C03630=1024.306,162.118,386.743,168.433,48.215,159.034
C03631=1024.301,161.869,386.765,168.430,48.220,159.035
C03632=1024.295,161.621,386.787,168.426,48.224,159.035
C03633=1024.290,161.372,386.809,168.423,48.229,159.036
C03634=1024.285,161.122,386.831,168.420,48.233,159.036
C03635=1024.279,160.874,386.853,168.417,48.238,159.037
C03636=1024.274,160.624,386.875,168.413,48.243,159.037
C03637=1024.269,160.375,386.897,168.410,48.247,159.037
C03638=1024.263,160.126,386.918,168.407,48.251,159.038
C03639=1024.258,159.878,386.941,168.403,48.256,159.038
C03640=1024.252,159.628,386.963,168.400,48.261,159.039
C03641=1024.247,159.380,386.985,168.397,48.265,159.039
C03642=1024.241,159.130,387.007,168.394,48.270,159.040
C03643=1024.236,158.882,387.028,168.391,48.275,159.040
C03644=1024.229,158.633,387.050,168.387,48.280,159.041
C03645=1024.225,158.383,387.071,168.384,48.285,159.041
C03646=1024.219,158.134,387.092,168.381,48.289,159.042
C03647=1024.213,157.886,387.114,168.378,48.294,159.042
C03648=1024.207,157.636,387.135,168.374,48.299,159.043
C03649=1024.202,157.388,387.157,168.371,48.303,159.043
C03650=1024.196,157.138,387.179,168.367,48.308,159.044
C03651=1024.190,156.890,387.200,168.365,48.313,159.044
C03652=1024.185,156.640,387.221,168.361,48.318,159.045
C03653=1024.179,156.392,387.242,168.358,48.322,159.045
C03654=1024.173,156.108,387.268,168.355,48.327,159.046
C03655=1024.166,155.825,387.292,168.350,48.333,159.046
C03656=1024.160,155.541,387.316,168.347,48.339,159.047
C03657=1024.153,155.258,387.340,168.343,48.344,159.047
C03658=1024.148,155.010,387.362,168.340,48.348,159.048
C03659=1024.142,154.760,387.383,168.337,48.353,159.048
C03660=1024.137,154.511,387.404,168.333,48.358,159.049
C03661=1024.131,154.262,387.426,168.330,48.363,159.049
C03662=1024.125,154.013,387.447,168.328,48.367,159.050
C03663=1024.119,153.764,387.468,168.324,48.372,159.050
C03664=1024.114,153.515,387.490,168.321,48.377,159.051
C03665=1024.109,153.266,387.511,168.317,48.382,159.051
C03666=1024.103,153.016,387.532,168.315,48.386,159.052
C03667=1024.098,152.768,387.554,168.311,48.391,159.052
C03668=1024.091,152.519,387.575,168.308,48.396,159.053
C03669=1024.086,152.270,387.596,168.305,48.401,159.053
C03670=1024.080,152.020,387.617,168.302,48.406,159.054
C03671=1024.074,151.772,387.639,168.299,48.411,159.054
C03672=1024.069,151.523,387.659,168.295,48.415,159.055
C03673=1024.063,151.274,387.681,168.292,48.420,159.055
C03674=1024.058,151.024,387.701,168.289,48.425,159.056
C03675=1024.052,150.775,387.723,168.286,48.430,159.056
C03676=1024.046,150.527,387.744,168.283,48.434,159.057
C03677=1024.041,150.278,387.765,168.279,48.439,159.057
C03678=1024.035,150.028,387.786,168.277,48.444,159.058
C03679=1024.029,149.779,387.807,168.273,48.449,159.058
C03680=1024.024,149.531,387.829,168.270,48.453,159.059
C03681=1024.019,149.281,387.850,168.266,48.458,159.059
C03682=1024.013,149.032,387.871,168.264,48.463,159.060
C03683=1024.008,148.783,387.892,168.260,48.468,159.060
C03684=1024.002,148.534,387.913,168.257,48.473,159.061
C03685=1023.996,148.285,387.934,168.255,48.477,159.061
C03686=1023.991,148.036,387.955,168.251,48.483,159.062
C03687=1023.985,147.786,387.976,168.248,48.487,159.063
C03688=1023.979,147.538,387.997,168.245,48.492,159.063
C03689=1023.974,147.289,388.018,168.242,48.497,159.064
C03690=1023.967,147.040,388.039,168.239,48.502,159.064
C03691=1023.962,146.791,388.059,168.235,48.506,159.065
C03692=1023.957,146.542,388.080,168.233,48.511,159.065
C03693=1023.951,146.292,388.102,168.229,48.516,159.066
C03694=1023.945,146.043,388.122,168.226,48.521,159.066
C03695=1023.940,145.795,388.143,168.224,48.525,159.067
C03696=1023.934,145.545,388.164,168.220,48.531,159.067
C03697=1023.929,145.296,388.185,168.217,48.536,159.068
C03698=1023.922,145.048,388.206,168.214,48.540,159.068
C03699=1023.917,144.799,388.226,168.211,48.545,159.069
C03700=1023.911,144.549,388.247,168.208,48.550,159.069
C03701=1023.906,144.300,388.268,168.204,48.555,159.070
C03702=1023.900,144.051,388.288,168.202,48.560,159.070
C03703=1023.894,143.802,388.309,168.199,48.565,159.071
C03704=1023.889,143.552,388.330,168.195,48.570,159.071
C03705=1023.883,143.303,388.350,168.192,48.574,159.072
C03706=1023.878,143.055,388.372,168.189,48.579,159.072
C03707=1023.871,142.805,388.392,168.186,48.584,159.073
C03708=1023.866,142.556,388.412,168.183,48.589,159.073
C03709=1023.861,142.307,388.433,168.181,48.594,159.074
C03710=1023.855,142.059,388.454,168.177,48.599,159.074
C03711=1023.848,141.809,388.475,168.174,48.604,159.075
C03712=1023.843,141.560,388.495,168.171,48.608,159.076
C03713=1023.838,141.311,388.516,168.168,48.613,159.076
C03714=1023.833,141.062,388.536,168.164,48.618,159.076
C03715=1023.826,140.813,388.557,168.162,48.623,159.077
C03716=1023.821,140.564,388.578,168.159,48.628,159.078
C03717=1023.815,140.315,388.598,168.155,48.633,159.078
C03718=1023.809,140.031,388.622,168.152,48.638,159.079
C03719=1023.802,139.748,388.645,168.149,48.644,159.079
C03720=1023.796,139.463,388.668,168.145,48.649,159.080
C03721=1023.790,139.180,388.692,168.142,48.655,159.080
C03722=1023.785,138.931,388.713,168.139,48.659,159.081
C03723=1023.779,138.682,388.733,168.136,48.664,159.081
C03724=1023.773,138.433,388.753,168.133,48.670,159.082
C03725=1023.768,138.184,388.774,168.130,48.674,159.083
C03726=1023.762,137.934,388.795,168.127,48.679,159.083
C03727=1023.756,137.686,388.815,168.123,48.684,159.084
C03728=1023.751,137.437,388.836,168.121,48.688,159.084
C03729=1023.745,137.188,388.856,168.118,48.694,159.085
C03730=1023.739,136.939,388.876,168.115,48.699,159.085
C03731=1023.733,136.690,388.896,168.112,48.703,159.086
C03732=1023.728,136.440,388.917,168.109,48.708,159.086
C03733=1023.723,136.190,388.937,168.106,48.714,159.087
C03734=1023.717,135.942,388.957,168.103,48.718,159.087
C03735=1023.711,135.693,388.978,168.100,48.723,159.088
C03736=1023.705,135.444,388.998,168.096,48.728,159.088
C03737=1023.700,135.195,389.018,168.094,48.733,159.089
C03738=1023.694,134.946,389.038,168.091,48.738,159.090
C03739=1023.688,134.696,389.059,168.087,48.743,159.090
C03740=1023.682,134.447,389.079,168.085,48.748,159.091
C03741=1023.677,134.198,389.099,168.082,48.753,159.091
C03742=1023.671,133.949,389.119,168.079,48.758,159.092
C03743=1023.666,133.700,389.140,168.076,48.763,159.092
C03744=1023.660,133.451,389.159,168.073,48.768,159.093
C03745=1023.655,133.202,389.180,168.070,48.772,159.093
C03746=1023.649,132.953,389.200,168.067,48.778,159.094
C03747=1023.644,132.704,389.220,168.064,48.783,159.094
C03748=1023.638,132.455,389.240,168.061,48.787,159.095
C03749=1023.632,132.205,389.261,168.058,48.792,159.095
C03750=1023.626,131.956,389.281,168.055,48.797,159.096
C03751=1023.621,131.706,389.301,168.053,48.802,159.097
C03752=1023.615,131.458,389.321,168.049,48.807,159.097
C03753=1023.609,131.208,389.341,168.047,48.812,159.098
C03754=1023.603,130.960,389.361,168.043,48.817,159.098
C03755=1023.598,130.711,389.382,168.040,48.822,159.099
C03756=1023.593,130.461,389.401,168.038,48.827,159.099
C03757=1023.587,130.212,389.421,168.034,48.832,159.100
C03758=1023.581,129.963,389.442,168.032,48.836,159.100
C03759=1023.576,129.714,389.461,168.029,48.842,159.101
C03760=1023.570,129.465,389.481,168.026,48.847,159.101
C03761=1023.564,129.216,389.501,168.023,48.851,159.102
C03762=1023.558,128.967,389.520,168.020,48.857,159.103
C03763=1023.553,128.718,389.541,168.017,48.862,159.103
C03764=1023.547,128.468,389.560,168.015,48.867,159.104
C03765=1023.540,128.219,389.580,168.011,48.872,159.104
C03766=1023.534,127.970,389.600,168.008,48.877,159.105
C03767=1023.529,127.720,389.619,168.006,48.882,159.105
C03768=1023.523,127.472,389.639,168.002,48.887,159.106
C03769=1023.517,127.222,389.659,167.999,48.892,159.106
C03770=1023.512,126.973,389.679,167.997,48.897,159.107
C03771=1023.506,126.724,389.698,167.994,48.902,159.108
C03772=1023.500,126.475,389.718,167.990,48.908,159.108
C03773=1023.494,126.225,389.738,167.988,48.912,159.109
C03774=1023.488,125.976,389.758,167.985,48.917,159.109
C03775=1023.483,125.727,389.777,167.982,48.923,159.110
C03776=1023.477,125.478,389.797,167.979,48.927,159.110
C03777=1023.471,125.229,389.817,167.976,48.932,159.111
C03778=1023.466,124.980,389.837,167.974,48.938,159.112
C03779=1023.460,124.730,389.856,167.970,48.942,159.112
C03780=1023.454,124.481,389.876,167.967,48.947,159.113
C03781=1023.448,124.232,389.895,167.965,48.953,159.113
C03782=1023.442,123.948,389.917,167.961,48.958,159.114
C03783=1023.435,123.665,389.940,167.958,48.964,159.114
C03784=1023.429,123.381,389.962,167.955,48.970,159.115
C03785=1023.422,123.097,389.984,167.952,48.975,159.116
C03786=1023.418,122.849,390.005,167.948,48.980,159.116
C03787=1023.412,122.600,390.024,167.946,48.985,159.117
C03788=1023.406,122.351,390.044,167.943,48.990,159.117
C03789=1023.400,122.101,390.063,167.939,48.995,159.118
C03790=1023.394,121.852,390.083,167.937,49.001,159.119
C03791=1023.389,121.603,390.102,167.934,49.005,159.119
C03792=1023.383,121.354,390.121,167.932,49.010,159.120
C03793=1023.377,121.105,390.141,167.928,49.015,159.120
C03794=1023.372,120.855,390.161,167.926,49.020,159.121
C03795=1023.366,120.606,390.180,167.923,49.025,159.121
C03796=1023.360,120.357,390.200,167.919,49.030,159.122
C03797=1023.355,120.107,390.220,167.917,49.035,159.122
C03798=1023.349,119.859,390.239,167.914,49.040,159.123
C03799=1023.343,119.610,390.259,167.912,49.045,159.123
C03800=1023.338,119.360,390.278,167.909,49.051,159.124
C03801=1023.332,119.112,390.298,167.906,49.055,159.125
C03802=1023.327,118.862,390.318,167.903,49.060,159.125
C03803=1023.321,118.612,390.337,167.900,49.065,159.126
C03804=1023.315,118.364,390.357,167.897,49.070,159.126
C03805=1023.309,118.114,390.376,167.894,49.075,159.127
C03806=1023.304,117.865,390.395,167.892,49.080,159.127
C03807=1023.299,117.616,390.414,167.888,49.085,159.128
C03808=1023.293,117.367,390.434,167.886,49.090,159.128
C03809=1023.287,117.118,390.453,167.883,49.095,159.129
C03810=1023.281,116.868,390.473,167.881,49.100,159.130
C03811=1023.276,116.619,390.493,167.877,49.104,159.130
C03812=1023.271,116.370,390.512,167.875,49.110,159.131
C03813=1023.265,116.121,390.531,167.872,49.115,159.131
C03814=1023.260,115.872,390.550,167.869,49.119,159.132
C03815=1023.254,115.623,390.570,167.866,49.124,159.132
C03816=1023.248,115.373,390.590,167.864,49.130,159.133
C03817=1023.243,115.125,390.609,167.861,49.135,159.133
C03818=1023.237,114.875,390.628,167.858,49.139,159.134
C03819=1023.231,114.626,390.647,167.855,49.144,159.134
C03820=1023.226,114.377,390.668,167.853,49.149,159.135
C03821=1023.220,114.127,390.687,167.849,49.154,159.136
C03822=1023.215,113.878,390.706,167.847,49.159,159.136
C03823=1023.210,113.629,390.725,167.844,49.164,159.137
C03824=1023.204,113.380,390.744,167.841,49.168,159.137
C03825=1023.198,113.131,390.764,167.838,49.174,159.138
C03826=1023.193,112.882,390.783,167.836,49.179,159.138
C03827=1023.187,112.633,390.802,167.833,49.184,159.139
C03828=1023.182,112.383,390.822,167.830,49.188,159.139
C03829=1023.176,112.134,390.841,167.827,49.194,159.140
C03830=1023.170,111.884,390.860,167.825,49.199,159.140
C03831=1023.165,111.636,390.879,167.821,49.203,159.141
C03832=1023.159,111.386,390.898,167.819,49.209,159.142
C03833=1023.153,111.137,390.917,167.816,49.214,159.142
C03834=1023.147,110.888,390.936,167.814,49.219,159.143
C03835=1023.142,110.639,390.955,167.811,49.224,159.143
C03836=1023.137,110.389,390.974,167.808,49.229,159.144
C03837=1023.131,110.140,390.993,167.805,49.234,159.144
C03838=1023.124,109.891,391.012,167.802,49.239,159.145
C03839=1023.119,109.642,391.031,167.800,49.244,159.145
C03840=1023.114,109.393,391.050,167.797,49.249,159.146
C03841=1023.107,109.144,391.069,167.794,49.254,159.147
C03842=1023.102,108.894,391.088,167.791,49.260,159.147
C03843=1023.097,108.645,391.106,167.789,49.264,159.148
C03844=1023.090,108.396,391.125,167.785,49.269,159.148
C03845=1023.085,108.146,391.144,167.783,49.275,159.149
C03846=1023.078,107.862,391.166,167.779,49.281,159.150
C03847=1023.072,107.579,391.187,167.776,49.286,159.150
C03848=1023.065,107.295,391.209,167.773,49.292,159.151
C03849=1023.058,107.011,391.230,167.770,49.298,159.151
C03850=1023.053,106.762,391.249,167.767,49.303,159.152
C03851=1023.047,106.513,391.267,167.765,49.308,159.153
C03852=1023.041,106.264,391.286,167.762,49.313,159.153
C03853=1023.036,106.014,391.306,167.760,49.318,159.154
C03854=1023.030,105.765,391.323,167.756,49.323,159.154
C03855=1023.024,105.516,391.343,167.754,49.328,159.155
C03856=1023.018,105.267,391.361,167.751,49.333,159.155
C03857=1023.013,105.018,391.380,167.749,49.339,159.156
C03858=1023.008,104.768,391.399,167.746,49.344,159.157
C03859=1023.001,104.519,391.417,167.743,49.348,159.157
C03860=1022.996,104.270,391.436,167.740,49.354,159.158
C03861=1022.990,104.021,391.455,167.738,49.359,159.158
C03862=1022.984,103.771,391.473,167.734,49.364,159.159
C03863=1022.979,103.522,391.492,167.731,49.369,159.159
C03864=1022.973,103.273,391.511,167.729,49.374,159.160
C03865=1022.967,103.024,391.530,167.726,49.379,159.160
C03866=1022.962,102.774,391.548,167.724,49.384,159.161
C03867=1022.956,102.525,391.567,167.721,49.389,159.162
C03868=1022.950,102.276,391.586,167.718,49.394,159.162
C03869=1022.945,102.027,391.605,167.716,49.399,159.163
C03870=1022.939,101.777,391.623,167.713,49.404,159.163
C03871=1022.934,101.529,391.642,167.710,49.409,159.164
C03872=1022.927,101.279,391.660,167.707,49.414,159.165
C03873=1022.922,101.029,391.679,167.705,49.419,159.165
C03874=1022.917,100.781,391.698,167.702,49.424,159.166
C03875=1022.910,100.532,391.717,167.700,49.429,159.166
C03876=1022.906,100.282,391.735,167.696,49.434,159.167
C03877=1022.900,100.033,391.754,167.694,49.439,159.167
C03878=1022.894,99.783,391.772,167.691,49.445,159.168
C03879=1022.889,99.534,391.791,167.689,49.449,159.168
C03880=1022.882,99.285,391.809,167.685,49.454,159.169
C03881=1022.877,99.035,391.828,167.683,49.460,159.170
C03882=1022.871,98.787,391.846,167.680,49.465,159.170
C03883=1022.865,98.537,391.864,167.678,49.470,159.171
C03884=1022.860,98.288,391.883,167.675,49.475,159.171
C03885=1022.854,98.039,391.901,167.673,49.480,159.172
C03886=1022.847,97.789,391.920,167.669,49.485,159.172
C03887=1022.843,97.540,391.938,167.666,49.490,159.173
C03888=1022.836,97.291,391.956,167.664,49.496,159.174
C03889=1022.831,97.042,391.974,167.661,49.501,159.174
C03890=1022.825,96.792,391.992,167.659,49.506,159.175
C03891=1022.819,96.543,392.011,167.655,49.511,159.175
C03892=1022.813,96.294,392.029,167.653,49.516,159.176
C03893=1022.808,96.044,392.048,167.650,49.521,159.176
C03894=1022.802,95.795,392.066,167.648,49.526,159.177
C03895=1022.796,95.546,392.084,167.645,49.532,159.178
C03896=1022.791,95.297,392.102,167.642,49.536,159.178
C03897=1022.785,95.047,392.120,167.639,49.542,159.179
C03898=1022.779,94.799,392.139,167.637,49.547,159.179
C03899=1022.774,94.548,392.157,167.634,49.552,159.180
C03900=1022.768,94.300,392.175,167.632,49.557,159.181
C03901=1022.762,94.050,392.193,167.628,49.562,159.181
C03902=1022.756,93.801,392.211,167.626,49.567,159.182
C03903=1022.750,93.552,392.230,167.623,49.572,159.182
C03904=1022.745,93.303,392.248,167.621,49.577,159.183
C03905=1022.739,93.053,392.266,167.618,49.583,159.183
C03906=1022.734,92.804,392.284,167.616,49.587,159.184
C03907=1022.728,92.555,392.302,167.612,49.592,159.184
C03908=1022.722,92.306,392.321,167.610,49.598,159.185
C03909=1022.716,92.056,392.339,167.607,49.603,159.185
C03910=1022.710,91.773,392.360,167.604,49.608,159.186
C03911=1022.703,91.488,392.380,167.601,49.614,159.187
C03912=1022.697,91.205,392.401,167.598,49.620,159.187
C03913=1022.691,90.922,392.421,167.595,49.625,159.188
C03914=1022.684,90.672,392.439,167.593,49.631,159.189
C03915=1022.679,90.423,392.458,167.590,49.636,159.189
C03916=1022.673,90.174,392.476,167.587,49.640,159.190
C03917=1022.668,89.925,392.494,167.584,49.646,159.190
C03918=1022.662,89.674,392.512,167.582,49.651,159.191
C03919=1022.657,89.426,392.531,167.579,49.656,159.191
C03920=1022.651,89.177,392.548,167.577,49.661,159.192
C03921=1022.645,88.927,392.566,167.573,49.666,159.193
C03922=1022.639,88.678,392.584,167.571,49.672,159.193
C03923=1022.633,88.428,392.602,167.568,49.677,159.194
C03924=1022.628,88.179,392.619,167.566,49.682,159.194
C03925=1022.622,87.930,392.637,167.563,49.687,159.195
C03926=1022.616,87.681,392.655,167.561,49.692,159.196
C03927=1022.610,87.432,392.673,167.558,49.697,159.196
C03928=1022.604,87.183,392.691,167.555,49.702,159.197
C03929=1022.598,86.933,392.709,167.552,49.708,159.197
C03930=1022.593,86.684,392.726,167.550,49.712,159.198
C03931=1022.587,86.435,392.744,167.547,49.718,159.198
C03932=1022.581,86.185,392.762,167.545,49.723,159.199
C03933=1022.575,85.936,392.779,167.542,49.728,159.200
C03934=1022.569,85.686,392.797,167.539,49.733,159.200
C03935=1022.564,85.437,392.815,167.536,49.739,159.201
C03936=1022.558,85.187,392.833,167.534,49.744,159.201
C03937=1022.552,84.938,392.850,167.531,49.749,159.202
C03938=1022.547,84.689,392.868,167.529,49.754,159.202
C03939=1022.540,84.440,392.886,167.526,49.759,159.203
C03940=1022.535,84.191,392.903,167.524,49.764,159.204
C03941=1022.529,83.941,392.921,167.520,49.769,159.204
C03942=1022.523,83.692,392.939,167.518,49.774,159.205
C03943=1022.518,83.443,392.957,167.515,49.780,159.205
C03944=1022.512,83.193,392.974,167.513,49.784,159.206
C03945=1022.506,82.944,392.992,167.510,49.790,159.206
C03946=1022.501,82.695,393.010,167.508,49.795,159.207
C03947=1022.495,82.445,393.028,167.504,49.800,159.207
C03948=1022.489,82.196,393.045,167.502,49.805,159.208
C03949=1022.483,81.947,393.063,167.499,49.810,159.209
C03950=1022.477,81.697,393.081,167.497,49.816,159.209
C03951=1022.472,81.448,393.098,167.494,49.821,159.210
C03952=1022.466,81.199,393.116,167.491,49.825,159.210
C03953=1022.460,80.950,393.134,167.489,49.831,159.211
C03954=1022.455,80.700,393.151,167.486,49.836,159.211
C03955=1022.449,80.451,393.169,167.484,49.841,159.212
C03956=1022.443,80.202,393.187,167.481,49.846,159.213
C03957=1022.438,79.952,393.204,167.479,49.851,159.213
C03958=1022.432,79.703,393.221,167.475,49.856,159.214
C03959=1022.426,79.453,393.239,167.473,49.861,159.214
C03960=1022.421,79.204,393.257,167.470,49.866,159.215
C03961=1022.415,78.955,393.274,167.468,49.871,159.215
C03962=1022.409,78.705,393.292,167.465,49.877,159.216
C03963=1022.404,78.456,393.310,167.463,49.882,159.216
C03964=1022.398,78.207,393.327,167.460,49.886,159.217
C03965=1022.392,77.958,393.345,167.457,49.891,159.217
C03966=1022.387,77.708,393.362,167.455,49.897,159.218
C03967=1022.381,77.459,393.380,167.452,49.902,159.219
C03968=1022.376,77.210,393.397,167.449,49.906,159.219
C03969=1022.369,76.960,393.415,167.446,49.912,159.220
C03970=1022.364,76.711,393.431,167.444,49.917,159.220
C03971=1022.358,76.462,393.449,167.441,49.923,159.221
C03972=1022.353,76.213,393.467,167.439,49.927,159.222
C03973=1022.346,75.963,393.484,167.436,49.932,159.222
C03974=1022.340,75.679,393.504,167.433,49.939,159.223
C03975=1022.333,75.396,393.524,167.430,49.945,159.223
C03976=1022.327,75.112,393.543,167.427,49.950,159.224
C03977=1022.320,74.828,393.562,167.424,49.956,159.225
C03978=1022.314,74.579,393.580,167.421,49.962,159.225
C03979=1022.309,74.330,393.597,167.419,49.966,159.226
C03980=1022.302,74.080,393.614,167.417,49.971,159.226
C03981=1022.297,73.831,393.632,167.414,49.977,159.227
C03982=1022.292,73.582,393.649,167.411,49.982,159.228
C03983=1022.285,73.333,393.666,167.409,49.987,159.228
C03984=1022.279,73.083,393.684,167.406,49.992,159.229
C03985=1022.274,72.833,393.700,167.403,49.997,159.229
C03986=1022.268,72.584,393.718,167.401,50.003,159.230
C03987=1022.262,72.335,393.734,167.398,50.008,159.230
C03988=1022.256,72.085,393.752,167.395,50.012,159.231
C03989=1022.251,71.836,393.770,167.393,50.018,159.231
C03990=1022.245,71.587,393.786,167.390,50.023,159.232
C03991=1022.239,71.338,393.803,167.387,50.028,159.232
C03992=1022.234,71.088,393.820,167.385,50.033,159.233
C03993=1022.227,70.839,393.838,167.382,50.038,159.234
C03994=1022.222,70.589,393.855,167.380,50.044,159.234
C03995=1022.217,70.340,393.872,167.377,50.049,159.235
C03996=1022.211,70.091,393.888,167.374,50.053,159.235
C03997=1022.205,69.842,393.906,167.372,50.059,159.236
C03998=1022.200,69.593,393.923,167.369,50.064,159.236
C03999=1022.193,69.343,393.940,167.367,50.069,159.237
C04000=1022.188,69.094,393.958,167.364,50.074,159.238
C04001=1022.182,68.844,393.975,167.362,50.079,159.238
C04002=1022.176,68.595,393.992,167.358,50.084,159.239
C04003=1022.171,68.346,394.008,167.356,50.090,159.239
C04004=1022.164,68.095,394.025,167.353,50.095,159.240
C04005=1022.159,67.846,394.043,167.351,50.099,159.240
C04006=1022.153,67.597,394.059,167.348,50.105,159.241
C04007=1022.147,67.348,394.076,167.346,50.110,159.242
C04008=1022.141,67.099,394.093,167.343,50.116,159.242
C04009=1022.136,66.850,394.110,167.340,50.120,159.243
C04010=1022.130,66.600,394.126,167.337,50.125,159.243
C04011=1022.124,66.350,394.144,167.335,50.131,159.244
C04012=1022.118,66.101,394.161,167.332,50.136,159.244
C04013=1022.113,65.852,394.177,167.330,50.141,159.245
C04014=1022.107,65.602,394.194,167.327,50.146,159.245
C04015=1022.101,65.353,394.211,167.325,50.151,159.246
C04016=1022.095,65.104,394.228,167.323,50.157,159.247
C04017=1022.090,64.854,394.244,167.319,50.162,159.247
C04018=1022.084,64.605,394.261,167.317,50.166,159.248
C04019=1022.078,64.355,394.279,167.314,50.172,159.248
C04020=1022.072,64.106,394.295,167.312,50.177,159.249
C04021=1022.066,63.857,394.312,167.309,50.182,159.249
C04022=1022.060,63.607,394.329,167.307,50.187,159.250
C04023=1022.055,63.358,394.346,167.303,50.193,159.250
C04024=1022.049,63.108,394.362,167.301,50.197,159.251
C04025=1022.043,62.860,394.379,167.298,50.203,159.252
C04026=1022.037,62.610,394.395,167.296,50.208,159.252
C04027=1022.031,62.360,394.412,167.293,50.214,159.253
C04028=1022.025,62.111,394.429,167.291,50.218,159.253
C04029=1022.019,61.861,394.445,167.288,50.224,159.254
C04030=1022.013,61.612,394.461,167.285,50.229,159.254
C04031=1022.007,61.362,394.477,167.283,50.235,159.255
C04032=1022.001,61.114,394.494,167.280,50.240,159.256
C04033=1021.996,60.864,394.511,167.278,50.245,159.256
C04034=1021.990,60.615,394.527,167.274,50.250,159.257
C04035=1021.984,60.365,394.544,167.273,50.256,159.257
C04036=1021.978,60.116,394.560,167.269,50.261,159.258
C04037=1021.972,59.867,394.576,167.267,50.266,159.259
C04038=1021.965,59.549,394.597,167.264,50.273,159.259
C04039=1021.957,59.232,394.618,167.260,50.280,159.260
C04040=1021.950,58.915,394.638,167.257,50.287,159.261
C04041=1021.942,58.598,394.660,167.254,50.293,159.262
C04042=1021.937,58.348,394.677,167.251,50.298,159.262
C04043=1021.931,58.099,394.693,167.248,50.304,159.263
C04044=1021.924,57.849,394.710,167.246,50.309,159.263
C04045=1021.918,57.599,394.726,167.242,50.314,159.264
C04046=1021.912,57.350,394.742,167.241,50.319,159.264
C04047=1021.906,57.101,394.758,167.237,50.324,159.265
C04048=1021.900,56.851,394.775,167.235,50.330,159.265
C04049=1021.895,56.602,394.791,167.232,50.335,159.266
C04050=1021.889,56.352,394.808,167.230,50.340,159.266
C04051=1021.883,56.103,394.824,167.227,50.345,159.267
C04052=1021.877,55.854,394.840,167.225,50.350,159.268
C04053=1021.871,55.604,394.856,167.222,50.356,159.268
C04054=1021.865,55.355,394.873,167.220,50.361,159.269
C04055=1021.859,55.106,394.889,167.216,50.366,159.269
C04056=1021.854,54.856,394.906,167.215,50.371,159.270
C04057=1021.848,54.607,394.922,167.211,50.376,159.270
C04058=1021.843,54.358,394.938,167.209,50.381,159.271
C04059=1021.837,54.109,394.954,167.206,50.387,159.271
C04060=1021.831,53.859,394.970,167.204,50.392,159.272
C04061=1021.825,53.609,394.986,167.201,50.397,159.273
C04062=1021.819,53.360,395.002,167.199,50.402,159.273
C04063=1021.813,53.111,395.019,167.196,50.407,159.274
C04064=1021.808,52.861,395.035,167.194,50.413,159.274
C04065=1021.802,52.612,395.052,167.190,50.418,159.275
C04066=1021.796,52.362,395.068,167.188,50.423,159.275
C04067=1021.790,52.113,395.084,167.185,50.428,159.276
C04068=1021.784,51.864,395.100,167.183,50.433,159.276
C04069=1021.778,51.614,395.117,167.180,50.438,159.277
C04070=1021.774,51.381,395.132,167.178,50.443,159.277
C04071=1021.768,51.149,395.147,167.175,50.448,159.278
C04072=1021.763,50.916,395.162,167.173,50.453,159.278
C04073=1021.757,50.684,395.177,167.171,50.457,159.279
C04074=1021.752,50.450,395.192,167.169,50.462,159.280
C04075=1021.747,50.218,395.207,167.165,50.467,159.280
C04076=1021.742,49.985,395.222,167.163,50.472,159.280
C04077=1021.736,49.752,395.237,167.161,50.476,159.281
C04078=1021.730,49.503,395.253,167.159,50.482,159.282
C04079=1021.725,49.254,395.269,167.155,50.487,159.282
C04080=1021.719,49.005,395.286,167.153,50.492,159.283
C04081=1021.713,48.756,395.302,167.150,50.497,159.283
C04082=1021.708,48.505,395.318,167.148,50.502,159.284
C04083=1021.702,48.256,395.334,167.145,50.507,159.284
C04084=1021.696,48.007,395.350,167.143,50.512,159.285
C04085=1021.690,47.757,395.367,167.140,50.517,159.285
C04086=1021.684,47.509,395.383,167.137,50.523,159.286
C04087=1021.679,47.259,395.398,167.135,50.527,159.286
C04088=1021.673,47.009,395.414,167.132,50.533,159.287
C04089=1021.667,46.760,395.431,167.130,50.537,159.287
C04090=1021.661,46.511,395.447,167.127,50.542,159.288
C04091=1021.656,46.260,395.463,167.125,50.548,159.288
C04092=1021.651,46.012,395.479,167.122,50.553,159.289
C04093=1021.645,45.762,395.495,167.119,50.558,159.289
C04094=1021.639,45.513,395.511,167.117,50.563,159.290
C04095=1021.633,45.263,395.527,167.114,50.568,159.290
C04096=1021.627,45.014,395.543,167.112,50.572,159.291
C04097=1021.622,44.765,395.559,167.109,50.578,159.292
C04098=1021.616,44.516,395.575,167.106,50.583,159.292
C04099=1021.610,44.266,395.591,167.104,50.588,159.293
C04100=1021.604,44.016,395.607,167.101,50.593,159.293
C04101=1021.599,43.767,395.624,167.099,50.598,159.294
C04102=1021.593,43.483,395.641,167.096,50.604,159.294
C04103=1021.586,43.199,395.660,167.093,50.609,159.295
C04104=1021.580,42.914,395.678,167.090,50.615,159.295
C04105=1021.574,42.631,395.696,167.087,50.620,159.296
C04106=1021.568,42.382,395.713,167.084,50.626,159.296
C04107=1021.562,42.132,395.728,167.082,50.631,159.297
C04108=1021.556,41.883,395.744,167.079,50.636,159.297
C04109=1021.551,41.633,395.759,167.076,50.641,159.298
C04110=1021.545,41.384,395.775,167.074,50.647,159.299
C04111=1021.539,41.134,395.791,167.071,50.652,159.299
C04112=1021.532,40.885,395.807,167.068,50.657,159.299
C04113=1021.527,40.636,395.822,167.066,50.661,159.300
C04114=1021.521,40.386,395.838,167.063,50.667,159.301
C04115=1021.516,40.136,395.854,167.061,50.672,159.301
C04116=1021.510,39.887,395.870,167.058,50.677,159.302
C04117=1021.505,39.638,395.885,167.055,50.682,159.302
C04118=1021.498,39.388,395.900,167.052,50.688,159.303
C04119=1021.492,39.139,395.916,167.050,50.693,159.303
C04120=1021.487,38.889,395.932,167.047,50.698,159.304
C04121=1021.481,38.640,395.948,167.045,50.703,159.304
C04122=1021.476,38.390,395.963,167.042,50.708,159.305
C04123=1021.469,38.141,395.979,167.040,50.713,159.305
C04124=1021.463,37.891,395.994,167.038,50.718,159.306
C04125=1021.458,37.643,396.010,167.034,50.723,159.306
C04126=1021.452,37.393,396.026,167.032,50.728,159.307
C04127=1021.447,37.143,396.041,167.029,50.733,159.307
C04128=1021.441,36.894,396.057,167.027,50.739,159.308
C04129=1021.435,36.644,396.072,167.024,50.744,159.308
C04130=1021.429,36.394,396.088,167.022,50.749,159.309
C04131=1021.423,36.145,396.103,167.018,50.754,159.309
C04132=1021.418,35.896,396.119,167.017,50.759,159.310
C04133=1021.412,35.646,396.134,167.013,50.764,159.311
C04134=1021.406,35.396,396.149,167.011,50.769,159.311
C04135=1021.400,35.148,396.165,167.008,50.775,159.312
C04136=1021.394,34.898,396.180,167.006,50.780,159.312
C04137=1021.388,34.648,396.195,167.003,50.785,159.313
C04138=1021.382,34.399,396.210,167.000,50.790,159.313
C04139=1021.376,34.150,396.226,166.998,50.796,159.314
C04140=1021.371,33.900,396.242,166.995,50.801,159.314
C04141=1021.365,33.651,396.256,166.992,50.806,159.315
C04142=1021.359,33.401,396.272,166.990,50.811,159.315
C04143=1021.353,33.152,396.288,166.987,50.816,159.316
C04144=1021.348,32.903,396.303,166.984,50.821,159.316
C04145=1021.341,32.653,396.318,166.982,50.826,159.317
C04146=1021.336,32.403,396.333,166.979,50.831,159.317
C04147=1021.330,32.154,396.348,166.977,50.837,159.318
C04148=1021.324,31.904,396.363,166.974,50.842,159.318
C04149=1021.318,31.655,396.380,166.972,50.847,159.319
C04150=1021.312,31.406,396.394,166.968,50.852,159.319
C04151=1021.307,31.156,396.410,166.966,50.858,159.320
C04152=1021.301,30.907,396.424,166.963,50.863,159.320
C04153=1021.295,30.657,396.440,166.961,50.867,159.321
C04154=1021.289,30.407,396.455,166.958,50.873,159.321
C04155=1021.284,30.159,396.471,166.956,50.877,159.322
C04156=1021.277,29.909,396.486,166.953,50.883,159.323
C04157=1021.272,29.660,396.501,166.951,50.888,159.323
C04158=1021.267,29.410,396.516,166.947,50.893,159.324
C04159=1021.260,29.160,396.531,166.945,50.898,159.324
C04160=1021.255,28.911,396.546,166.942,50.903,159.324
C04161=1021.249,28.661,396.561,166.940,50.908,159.325
C04162=1021.244,28.412,396.577,166.937,50.913,159.325
C04163=1021.237,28.162,396.592,166.935,50.919,159.326
C04164=1021.232,27.912,396.607,166.932,50.924,159.327
C04165=1021.226,27.663,396.622,166.929,50.929,159.327
C04166=1021.219,27.379,396.639,166.927,50.935,159.328
C04167=1021.213,27.095,396.656,166.924,50.941,159.328
C04168=1021.206,26.811,396.673,166.920,50.947,159.329
C04169=1021.199,26.527,396.690,166.917,50.953,159.329
C04170=1021.194,26.277,396.705,166.915,50.957,159.330
C04171=1021.188,26.028,396.720,166.912,50.963,159.330
C04172=1021.182,25.779,396.735,166.909,50.967,159.331
C04173=1021.176,25.529,396.750,166.906,50.973,159.331
C04174=1021.170,25.279,396.765,166.904,50.978,159.332
C04175=1021.164,25.030,396.780,166.901,50.983,159.332
C04176=1021.159,24.780,396.795,166.899,50.988,159.333
C04177=1021.153,24.531,396.810,166.896,50.993,159.333
C04178=1021.147,24.282,396.825,166.893,50.999,159.334
C04179=1021.141,24.032,396.840,166.891,51.004,159.335
C04180=1021.135,23.782,396.854,166.888,51.009,159.335
C04181=1021.130,23.533,396.869,166.885,51.014,159.335
C04182=1021.123,23.284,396.884,166.882,51.019,159.336
C04183=1021.118,23.034,396.899,166.881,51.025,159.337
C04184=1021.112,22.785,396.914,166.877,51.030,159.337
C04185=1021.106,22.536,396.929,166.875,51.035,159.338
C04186=1021.100,22.286,396.944,166.872,51.040,159.338
C04187=1021.095,22.036,396.958,166.870,51.045,159.339
C04188=1021.089,21.786,396.973,166.867,51.050,159.339
C04189=1021.083,21.537,396.988,166.864,51.055,159.339
C04190=1021.077,21.288,397.003,166.862,51.061,159.340
C04191=1021.071,21.039,397.018,166.859,51.065,159.341
C04192=1021.066,20.789,397.032,166.856,51.071,159.341
C04193=1021.060,20.539,397.047,166.854,51.076,159.342
C04194=1021.054,20.290,397.062,166.851,51.081,159.342
C04195=1021.048,20.040,397.077,166.849,51.086,159.342
C04196=1021.043,19.791,397.092,166.845,51.091,159.343
C04197=1021.037,19.541,397.106,166.843,51.096,159.343
C04198=1021.031,19.292,397.121,166.840,51.101,159.344
C04199=1021.025,19.042,397.136,166.837,51.107,159.344
C04200=1021.020,18.792,397.150,166.835,51.111,159.345
C04201=1021.014,18.543,397.165,166.832,51.117,159.345
C04202=1021.008,18.294,397.180,166.830,51.122,159.346
C04203=1021.002,18.044,397.193,166.827,51.127,159.346
C04204=1020.996,17.795,397.208,166.825,51.132,159.347
C04205=1020.990,17.546,397.223,166.822,51.137,159.347
C04206=1020.984,17.295,397.237,166.819,51.142,159.348
C04207=1020.979,17.046,397.252,166.816,51.147,159.348
C04208=1020.973,16.797,397.267,166.814,51.152,159.349
C04209=1020.967,16.547,397.281,166.811,51.158,159.349
C04210=1020.961,16.298,397.296,166.808,51.163,159.350
C04211=1020.955,16.048,397.311,166.805,51.168,159.350
C04212=1020.950,15.799,397.325,166.803,51.173,159.351
C04213=1020.944,15.550,397.339,166.801,51.178,159.351
C04214=1020.938,15.299,397.354,166.797,51.183,159.352
C04215=1020.933,15.050,397.369,166.795,51.188,159.352
C04216=1020.927,14.801,397.382,166.792,51.194,159.353
C04217=1020.921,14.551,397.397,166.790,51.198,159.353
C04218=1020.915,14.302,397.412,166.787,51.204,159.354
C04219=1020.910,14.052,397.426,166.784,51.208,159.354
C04220=1020.903,13.803,397.441,166.781,51.214,159.355
C04221=1020.898,13.553,397.455,166.779,51.219,159.355
C04222=1020.892,13.303,397.470,166.776,51.224,159.356
C04223=1020.886,13.054,397.483,166.773,51.230,159.356
C04224=1020.880,12.805,397.498,166.771,51.234,159.357
C04225=1020.874,12.555,397.512,166.768,51.240,159.357
C04226=1020.868,12.305,397.526,166.766,51.245,159.358
C04227=1020.863,12.056,397.541,166.763,51.250,159.358
C04228=1020.857,11.806,397.555,166.760,51.256,159.359
C04229=1020.851,11.557,397.569,166.757,51.261,159.359
C04230=1020.844,11.274,397.585,166.755,51.266,159.360
C04231=1020.837,10.992,397.601,166.751,51.273,159.360
C04232=1020.831,10.709,397.617,166.748,51.279,159.361
C04233=1020.824,10.426,397.633,166.745,51.284,159.361
C04234=1020.818,10.177,397.647,166.742,51.290,159.362
C04235=1020.813,9.928,397.661,166.740,51.295,159.362
C04236=1020.806,9.678,397.675,166.737,51.300,159.363
C04237=1020.800,9.429,397.689,166.734,51.305,159.363
C04238=1020.795,9.179,397.703,166.731,51.310,159.364
C04239=1020.789,8.929,397.718,166.729,51.316,159.364
C04240=1020.783,8.680,397.732,166.727,51.321,159.365
C04241=1020.778,8.430,397.746,166.723,51.326,159.365
C04242=1020.772,8.181,397.760,166.720,51.331,159.366
C04243=1020.765,7.931,397.774,166.718,51.336,159.366
C04244=1020.759,7.682,397.788,166.715,51.341,159.367
C04245=1020.754,7.432,397.802,166.713,51.346,159.367
C04246=1020.749,7.183,397.816,166.710,51.351,159.368
C04247=1020.742,6.933,397.831,166.707,51.356,159.368
C04248=1020.737,6.683,397.845,166.705,51.362,159.369
C04249=1020.730,6.434,397.858,166.701,51.367,159.369
C04250=1020.725,6.185,397.872,166.699,51.372,159.370
C04251=1020.719,5.934,397.886,166.696,51.377,159.370
C04252=1020.713,5.685,397.901,166.694,51.382,159.371
C04253=1020.708,5.436,397.914,166.691,51.387,159.371
C04254=1020.702,5.186,397.928,166.688,51.393,159.371
C04255=1020.696,4.937,397.942,166.685,51.398,159.372
C04256=1020.690,4.687,397.957,166.682,51.403,159.372
C04257=1020.684,4.438,397.970,166.680,51.408,159.373
C04258=1020.679,4.188,397.984,166.677,51.413,159.373
C04259=1020.673,3.939,397.998,166.675,51.418,159.374
C04260=1020.668,3.689,398.012,166.672,51.423,159.374
C04261=1020.661,3.439,398.026,166.670,51.428,159.375
C04262=1020.655,3.190,398.040,166.666,51.433,159.375
C04263=1020.650,2.940,398.054,166.663,51.438,159.375
C04264=1020.644,2.691,398.068,166.661,51.443,159.376
C04265=1020.639,2.441,398.082,166.658,51.448,159.376
C04266=1020.633,2.192,398.096,166.656,51.453,159.377
C04267=1020.626,1.942,398.109,166.653,51.458,159.377
C04268=1020.621,1.692,398.123,166.650,51.463,159.378
C04269=1020.615,1.443,398.137,166.647,51.469,159.378
C04270=1020.610,1.194,398.152,166.645,51.473,159.379
C04271=1020.604,0.944,398.165,166.642,51.479,159.379
C04272=1020.598,0.695,398.179,166.639,51.484,159.380
C04273=1020.592,0.445,398.193,166.637,51.489,159.380
C04274=1020.587,0.196,398.206,166.634,51.494,159.380
C04275=1020.581,-0.055,398.221,166.631,51.499,159.381
C04276=1020.575,-0.304,398.235,166.628,51.504,159.381
C04277=1020.570,-0.554,398.248,166.626,51.509,159.382
C04278=1020.564,-0.803,398.262,166.623,51.514,159.382
C04279=1020.558,-1.053,398.276,166.620,51.518,159.383
C04280=1020.553,-1.302,398.289,166.617,51.524,159.383
C04281=1020.547,-1.552,398.303,166.615,51.529,159.384
C04282=1020.542,-1.801,398.317,166.612,51.534,159.384
C04283=1020.536,-2.051,398.330,166.610,51.539,159.384
C04284=1020.530,-2.300,398.344,166.607,51.544,159.385
C04285=1020.525,-2.550,398.358,166.605,51.549,159.385
C04286=1020.519,-2.799,398.372,166.601,51.553,159.386
C04287=1020.513,-3.050,398.386,166.598,51.559,159.386
C04288=1020.507,-3.299,398.399,166.596,51.564,159.387
C04289=1020.501,-3.548,398.413,166.593,51.569,159.387
C04290=1020.496,-3.798,398.427,166.590,51.574,159.387
C04291=1020.490,-4.048,398.441,166.587,51.579,159.388
C04292=1020.485,-4.297,398.455,166.585,51.584,159.388
C04293=1020.479,-4.546,398.468,166.582,51.589,159.389
C04294=1020.473,-4.827,398.483,166.579,51.594,159.389
C04295=1020.466,-5.108,398.498,166.576,51.600,159.390
C04296=1020.459,-5.389,398.513,166.573,51.606,159.390
C04297=1020.453,-5.670,398.528,166.569,51.612,159.391
C04298=1020.447,-5.919,398.541,166.567,51.617,159.391
C04299=1020.441,-6.168,398.555,166.564,51.623,159.392
C04300=1020.435,-6.418,398.568,166.561,51.628,159.392
C04301=1020.430,-6.668,398.582,166.559,51.633,159.393
C04302=1020.423,-6.917,398.595,166.556,51.638,159.393
C04303=1020.418,-7.167,398.609,166.554,51.643,159.394
C04304=1020.412,-7.416,398.622,166.551,51.648,159.394
C04305=1020.407,-7.666,398.635,166.547,51.653,159.394
C04306=1020.400,-7.915,398.648,166.545,51.658,159.395
C04307=1020.394,-8.165,398.662,166.542,51.664,159.395
C04308=1020.389,-8.415,398.675,166.539,51.669,159.396
C04309=1020.383,-8.664,398.688,166.537,51.674,159.396
C04310=1020.377,-8.914,398.702,166.533,51.678,159.396
C04311=1020.371,-9.164,398.715,166.531,51.683,159.397
C04312=1020.366,-9.413,398.728,166.528,51.688,159.397
C04313=1020.360,-9.662,398.742,166.525,51.694,159.398
C04314=1020.355,-9.913,398.755,166.523,51.699,159.398
C04315=1020.348,-10.162,398.768,166.520,51.704,159.399
C04316=1020.342,-10.411,398.781,166.517,51.709,159.399
C04317=1020.337,-10.661,398.795,166.514,51.714,159.400
C04318=1020.331,-10.911,398.808,166.511,51.719,159.400
C04319=1020.326,-11.160,398.821,166.509,51.724,159.400
C04320=1020.320,-11.409,398.834,166.506,51.730,159.401
C04321=1020.314,-11.659,398.848,166.503,51.735,159.401
C04322=1020.309,-11.909,398.860,166.501,51.740,159.402
C04323=1020.302,-12.158,398.874,166.498,51.745,159.402
C04324=1020.297,-12.408,398.887,166.495,51.749,159.402
C04325=1020.291,-12.658,398.900,166.492,51.754,159.403
C04326=1020.285,-12.907,398.914,166.489,51.760,159.403
C04327=1020.280,-13.157,398.926,166.487,51.765,159.404
C04328=1020.274,-13.407,398.940,166.484,51.770,159.404
C04329=1020.269,-13.656,398.952,166.481,51.775,159.405
C04330=1020.263,-13.905,398.966,166.478,51.780,159.405
C04331=1020.257,-14.155,398.979,166.476,51.784,159.405
C04332=1020.251,-14.405,398.992,166.473,51.790,159.406
C04333=1020.246,-14.655,399.005,166.470,51.795,159.406
C04334=1020.240,-14.904,399.019,166.467,51.800,159.407
C04335=1020.234,-15.154,399.031,166.464,51.805,159.407
C04336=1020.229,-15.403,399.045,166.462,51.809,159.407
C04337=1020.223,-15.653,399.057,166.459,51.814,159.408
C04338=1020.218,-15.902,399.071,166.456,51.820,159.408
C04339=1020.212,-16.152,399.084,166.453,51.825,159.409
C04340=1020.206,-16.401,399.097,166.450,51.830,159.409
C04341=1020.200,-16.651,399.109,166.447,51.835,159.409
C04342=1020.194,-16.901,399.122,166.445,51.840,159.410
C04343=1020.189,-17.150,399.135,166.442,51.845,159.410
C04344=1020.183,-17.400,399.148,166.439,51.851,159.411
C04345=1020.177,-17.650,399.161,166.437,51.856,159.411
C04346=1020.171,-17.899,399.174,166.434,51.861,159.412
C04347=1020.165,-18.149,399.186,166.430,51.866,159.412
C04348=1020.160,-18.398,399.199,166.428,51.871,159.413
C04349=1020.153,-18.647,399.212,166.425,51.876,159.413
C04350=1020.148,-18.898,399.225,166.422,51.881,159.413
C04351=1020.142,-19.147,399.237,166.420,51.886,159.414
C04352=1020.136,-19.397,399.250,166.416,51.891,159.414
C04353=1020.131,-19.646,399.263,166.413,51.896,159.414
C04354=1020.125,-19.896,399.276,166.411,51.901,159.415
C04355=1020.119,-20.146,399.288,166.408,51.907,159.415
C04356=1020.113,-20.396,399.301,166.406,51.912,159.416
C04357=1020.108,-20.644,399.314,166.403,51.917,159.416
C04358=1020.101,-20.923,399.328,166.400,51.922,159.417
C04359=1020.094,-21.203,399.342,166.397,51.928,159.417
C04360=1020.089,-21.481,399.356,166.393,51.934,159.418
C04361=1020.082,-21.761,399.371,166.390,51.939,159.418
C04362=1020.077,-22.010,399.383,166.388,51.944,159.418
C04363=1020.071,-22.259,399.396,166.384,51.949,159.419
C04364=1020.065,-22.509,399.409,166.381,51.955,159.419
C04365=1020.059,-22.758,399.421,166.379,51.959,159.420
C04366=1020.053,-23.008,399.434,166.376,51.965,159.420
C04367=1020.048,-23.258,399.446,166.373,51.969,159.420
C04368=1020.042,-23.508,399.459,166.371,51.974,159.421
C04369=1020.037,-23.757,399.472,166.367,51.980,159.421
C04370=1020.031,-24.007,399.485,166.364,51.985,159.422
C04371=1020.025,-24.257,399.497,166.362,51.989,159.422
C04372=1020.020,-24.506,399.509,166.359,51.994,159.422
C04373=1020.014,-24.756,399.522,166.357,51.999,159.423
C04374=1020.008,-25.006,399.535,166.353,52.005,159.423
C04375=1020.003,-25.255,399.547,166.350,52.010,159.424
C04376=1019.997,-25.505,399.560,166.348,52.014,159.424
C04377=1019.991,-25.755,399.572,166.345,52.019,159.424
C04378=1019.986,-26.003,399.585,166.343,52.024,159.425
C04379=1019.980,-26.253,399.598,166.340,52.030,159.425
C04380=1019.974,-26.503,399.610,166.336,52.034,159.425
C04381=1019.969,-26.752,399.623,166.334,52.039,159.426
C04382=1019.963,-27.002,399.635,166.331,52.045,159.426
C04383=1019.957,-27.252,399.648,166.327,52.049,159.426
C04384=1019.952,-27.502,399.661,166.325,52.054,159.427
C04385=1019.946,-27.752,399.673,166.322,52.059,159.427
C04386=1019.940,-28.001,399.685,166.320,52.064,159.428
C04387=1019.934,-28.250,399.697,166.317,52.070,159.428
C04388=1019.929,-28.501,399.709,166.314,52.075,159.429
C04389=1019.924,-28.750,399.721,166.310,52.079,159.429
C04390=1019.918,-29.000,399.734,166.308,52.084,159.429
C04391=1019.912,-29.250,399.746,166.305,52.090,159.430
C04392=1019.906,-29.499,399.759,166.302,52.095,159.430
C04393=1019.900,-29.748,399.771,166.300,52.100,159.431
C04394=1019.895,-29.998,399.783,166.297,52.105,159.431
C04395=1019.889,-30.248,399.795,166.294,52.111,159.431
C04396=1019.883,-30.498,399.807,166.291,52.115,159.432
C04397=1019.878,-30.747,399.819,166.288,52.120,159.432
C04398=1019.872,-30.997,399.832,166.285,52.125,159.432
C04399=1019.866,-31.246,399.843,166.282,52.131,159.433
C04400=1019.860,-31.496,399.856,166.280,52.136,159.433
C04401=1019.855,-31.745,399.868,166.276,52.140,159.433
C04402=1019.849,-31.996,399.880,166.273,52.146,159.434
C04403=1019.843,-32.245,399.893,166.271,52.151,159.434
C04404=1019.838,-32.495,399.905,166.268,52.156,159.435
C04405=1019.831,-32.744,399.917,166.265,52.161,159.435
C04406=1019.826,-32.994,399.928,166.262,52.165,159.435
C04407=1019.820,-33.244,399.941,166.259,52.171,159.436
C04408=1019.815,-33.493,399.953,166.256,52.176,159.436
C04409=1019.809,-33.743,399.965,166.254,52.181,159.437
C04410=1019.804,-33.993,399.977,166.251,52.186,159.437
C04411=1019.797,-34.242,399.989,166.247,52.191,159.437
C04412=1019.792,-34.491,400.001,166.245,52.196,159.438
C04413=1019.786,-34.741,400.014,166.242,52.201,159.438
C04414=1019.781,-34.991,400.025,166.239,52.206,159.438
C04415=1019.775,-35.241,400.038,166.237,52.211,159.439
C04416=1019.770,-35.490,400.050,166.234,52.216,159.439
C04417=1019.764,-35.740,400.061,166.230,52.221,159.439
C04418=1019.758,-35.990,400.073,166.228,52.226,159.440
C04419=1019.752,-36.239,400.086,166.225,52.231,159.440
C04420=1019.747,-36.489,400.098,166.221,52.236,159.440
C04421=1019.742,-36.738,400.110,166.219,52.241,159.441
C04422=1019.735,-37.017,400.123,166.216,52.246,159.441
C04423=1019.729,-37.294,400.136,166.213,52.251,159.442
C04424=1019.723,-37.573,400.149,166.209,52.258,159.442
C04425=1019.717,-37.850,400.163,166.206,52.263,159.443
C04426=1019.711,-38.100,400.175,166.204,52.267,159.443
C04427=1019.706,-38.350,400.187,166.201,52.273,159.443
C04428=1019.700,-38.600,400.199,166.198,52.278,159.444
C04429=1019.694,-38.849,400.211,166.195,52.282,159.444
C04430=1019.688,-39.099,400.223,166.192,52.287,159.444
C04431=1019.683,-39.349,400.235,166.189,52.293,159.445
C04432=1019.677,-39.598,400.246,166.186,52.297,159.445
C04433=1019.671,-39.848,400.258,166.183,52.302,159.445
C04434=1019.666,-40.098,400.270,166.180,52.308,159.446
C04435=1019.660,-40.347,400.282,166.177,52.313,159.446
C04436=1019.655,-40.597,400.293,166.175,52.318,159.447
C04437=1019.649,-40.847,400.304,166.172,52.323,159.447
C04438=1019.643,-41.096,400.317,166.168,52.328,159.447
C04439=1019.637,-41.346,400.327,166.166,52.333,159.448
C04440=1019.631,-41.596,400.340,166.163,52.338,159.448
C04441=1019.626,-41.845,400.351,166.160,52.343,159.448
C04442=1019.621,-42.095,400.362,166.157,52.348,159.449
C04443=1019.614,-42.345,400.374,166.155,52.353,159.449
C04444=1019.609,-42.595,400.386,166.152,52.359,159.449
C04445=1019.604,-42.844,400.398,166.148,52.363,159.450
C04446=1019.597,-43.094,400.409,166.146,52.368,159.450
C04447=1019.592,-43.344,400.421,166.143,52.373,159.451
C04448=1019.586,-43.593,400.432,166.139,52.378,159.451
C04449=1019.581,-43.843,400.444,166.136,52.383,159.451
C04450=1019.575,-44.093,400.455,166.134,52.388,159.452
C04451=1019.570,-44.342,400.467,166.131,52.393,159.452
C04452=1019.564,-44.591,400.478,166.128,52.398,159.452
C04453=1019.558,-44.842,400.490,166.126,52.403,159.453
C04454=1019.552,-45.091,400.501,166.122,52.408,159.453
C04455=1019.547,-45.340,400.513,166.119,52.413,159.453
C04456=1019.541,-45.591,400.524,166.117,52.418,159.454
C04457=1019.536,-45.840,400.536,166.113,52.423,159.454
C04458=1019.531,-46.090,400.548,166.110,52.428,159.454
C04459=1019.525,-46.339,400.559,166.108,52.433,159.455
C04460=1019.519,-46.590,400.571,166.105,52.438,159.455
C04461=1019.513,-46.838,400.582,166.102,52.443,159.455
C04462=1019.508,-47.088,400.594,166.100,52.448,159.456
C04463=1019.503,-47.338,400.604,166.096,52.453,159.456
C04464=1019.497,-47.588,400.616,166.093,52.458,159.456
C04465=1019.491,-47.838,400.627,166.090,52.463,159.456
C04466=1019.486,-48.087,400.639,166.088,52.468,159.457
C04467=1019.480,-48.336,400.650,166.085,52.473,159.457
C04468=1019.475,-48.587,400.662,166.081,52.478,159.457
C04469=1019.469,-48.836,400.673,166.079,52.483,159.458
C04470=1019.464,-49.086,400.684,166.075,52.487,159.458
C04471=1019.458,-49.335,400.696,166.073,52.492,159.459
C04472=1019.453,-49.585,400.708,166.070,52.497,159.459
C04473=1019.446,-49.835,400.719,166.067,52.502,159.459
C04474=1019.441,-50.085,400.730,166.064,52.507,159.459
C04475=1019.436,-50.334,400.741,166.061,52.512,159.460
C04476=1019.431,-50.584,400.753,166.058,52.517,159.460
C04477=1019.425,-50.833,400.764,166.056,52.522,159.460
C04478=1019.420,-51.083,400.776,166.053,52.527,159.461
C04479=1019.413,-51.333,400.787,166.049,52.532,159.461
C04480=1019.408,-51.583,400.797,166.046,52.537,159.461
C04481=1019.402,-51.833,400.808,166.043,52.542,159.462
C04482=1019.396,-52.082,400.819,166.041,52.547,159.462
C04483=1019.391,-52.332,400.830,166.038,52.553,159.463
C04484=1019.385,-52.581,400.841,166.034,52.557,159.463
C04485=1019.379,-52.832,400.852,166.031,52.563,159.463
C04486=1019.373,-53.110,400.864,166.029,52.569,159.464
C04487=1019.366,-53.387,400.876,166.026,52.574,159.464
C04488=1019.360,-53.666,400.889,166.021,52.580,159.464
C04489=1019.354,-53.944,400.900,166.018,52.585,159.465
C04490=1019.348,-54.194,400.911,166.015,52.591,159.465
C04491=1019.342,-54.443,400.922,166.012,52.596,159.465
C04492=1019.337,-54.693,400.934,166.010,52.601,159.466
C04493=1019.331,-54.943,400.945,166.007,52.606,159.466
C04494=1019.325,-55.193,400.955,166.004,52.611,159.466
C04495=1019.320,-55.443,400.966,166.001,52.616,159.467
C04496=1019.314,-55.692,400.977,165.997,52.621,159.467
C04497=1019.308,-55.942,400.988,165.995,52.626,159.467
C04498=1019.302,-56.191,400.999,165.992,52.631,159.468
C04499=1019.297,-56.442,401.009,165.989,52.637,159.468
C04500=1019.291,-56.691,401.020,165.985,52.641,159.468
C04501=1019.286,-56.941,401.031,165.983,52.646,159.469
C04502=1019.281,-57.190,401.042,165.980,52.652,159.469
C04503=1019.275,-57.440,401.053,165.977,52.657,159.469
C04504=1019.269,-57.690,401.063,165.974,52.662,159.470
C04505=1019.264,-57.939,401.074,165.972,52.667,159.470
C04506=1019.258,-58.189,401.085,165.968,52.672,159.470
C04507=1019.252,-58.438,401.096,165.965,52.677,159.471
C04508=1019.247,-58.688,401.106,165.962,52.682,159.471
C04509=1019.241,-58.938,401.117,165.960,52.687,159.471
C04510=1019.235,-59.187,401.128,165.957,52.692,159.472
C04511=1019.231,-59.438,401.138,165.954,52.697,159.472
C04512=1019.225,-59.687,401.149,165.950,52.702,159.472
C04513=1019.219,-59.937,401.160,165.948,52.707,159.473
C04514=1019.213,-60.186,401.171,165.945,52.712,159.473
C04515=1019.208,-60.436,401.181,165.941,52.717,159.473
C04516=1019.202,-60.686,401.192,165.938,52.722,159.474
C04517=1019.196,-60.935,401.203,165.936,52.727,159.474
C04518=1019.191,-61.186,401.213,165.933,52.732,159.474
C04519=1019.185,-61.435,401.224,165.929,52.737,159.475
C04520=1019.180,-61.685,401.234,165.926,52.742,159.475
C04521=1019.174,-61.935,401.245,165.924,52.747,159.475
C04522=1019.168,-62.184,401.256,165.921,52.752,159.476
C04523=1019.164,-62.435,401.267,165.918,52.757,159.476
C04524=1019.158,-62.684,401.277,165.914,52.762,159.476
C04525=1019.152,-62.934,401.288,165.912,52.767,159.477
C04526=1019.147,-63.184,401.299,165.909,52.772,159.477
C04527=1019.141,-63.433,401.309,165.906,52.777,159.477
C04528=1019.136,-63.683,401.320,165.903,52.782,159.477
C04529=1019.130,-63.933,401.330,165.900,52.787,159.478
C04530=1019.125,-64.182,401.340,165.897,52.792,159.478
C04531=1019.119,-64.432,401.351,165.894,52.797,159.478
C04532=1019.113,-64.681,401.362,165.892,52.802,159.479
C04533=1019.108,-64.931,401.372,165.888,52.806,159.479
C04534=1019.102,-65.181,401.383,165.885,52.812,159.479
C04535=1019.097,-65.431,401.393,165.882,52.816,159.479
C04536=1019.091,-65.680,401.404,165.880,52.822,159.480
C04537=1019.086,-65.931,401.415,165.876,52.826,159.480
C04538=1019.081,-66.180,401.425,165.873,52.832,159.480
C04539=1019.076,-66.430,401.435,165.871,52.836,159.481
C04540=1019.070,-66.679,401.446,165.868,52.841,159.481
C04541=1019.065,-66.929,401.457,165.864,52.846,159.481
C04542=1019.059,-67.179,401.467,165.861,52.851,159.482
C04543=1019.054,-67.429,401.478,165.859,52.856,159.482
C04544=1019.049,-67.678,401.487,165.856,52.861,159.482
C04545=1019.043,-67.928,401.498,165.852,52.866,159.482
C04546=1019.038,-68.178,401.508,165.850,52.871,159.483
C04547=1019.032,-68.427,401.519,165.847,52.875,159.483
C04548=1019.026,-68.677,401.529,165.843,52.880,159.483
C04549=1019.021,-68.926,401.540,165.840,52.886,159.483
C04550=1019.016,-69.206,401.551,165.837,52.891,159.484
C04551=1019.010,-69.486,401.563,165.834,52.896,159.484
C04552=1019.003,-69.765,401.575,165.831,52.902,159.485
C04553=1018.997,-70.045,401.587,165.827,52.907,159.485
C04554=1018.992,-70.294,401.596,165.824,52.912,159.485
C04555=1018.986,-70.544,401.607,165.821,52.917,159.485
C04556=1018.981,-70.794,401.618,165.818,52.922,159.485
C04557=1018.975,-71.044,401.628,165.815,52.926,159.486
C04558=1018.970,-71.293,401.638,165.812,52.932,159.486
C04559=1018.965,-71.543,401.648,165.809,52.936,159.486
C04560=1018.959,-71.793,401.659,165.807,52.941,159.487
C04561=1018.954,-72.043,401.669,165.803,52.946,159.487
C04562=1018.950,-72.292,401.680,165.800,52.951,159.487
C04563=1018.944,-72.542,401.690,165.798,52.956,159.488
C04564=1018.938,-72.792,401.701,165.794,52.960,159.488
C04565=1018.934,-73.041,401.711,165.791,52.965,159.488
C04566=1018.928,-73.291,401.721,165.789,52.970,159.488
C04567=1018.923,-73.541,401.731,165.786,52.975,159.488
C04568=1018.918,-73.790,401.741,165.782,52.980,159.489
C04569=1018.912,-74.040,401.752,165.780,52.985,159.489
C04570=1018.907,-74.290,401.762,165.777,52.989,159.489
C04571=1018.901,-74.541,401.772,165.774,52.995,159.490
C04572=1018.896,-74.789,401.782,165.770,52.999,159.490
C04573=1018.890,-75.039,401.792,165.768,53.004,159.490
C04574=1018.884,-75.289,401.802,165.765,53.009,159.490
C04575=1018.880,-75.539,401.812,165.762,53.015,159.491
C04576=1018.873,-75.788,401.822,165.758,53.019,159.491
C04577=1018.868,-76.039,401.832,165.756,53.024,159.491
C04578=1018.863,-76.288,401.842,165.753,53.030,159.492
C04579=1018.858,-76.538,401.852,165.750,53.034,159.492
C04580=1018.852,-76.787,401.861,165.747,53.040,159.492
C04581=1018.847,-77.037,401.871,165.744,53.044,159.492
C04582=1018.841,-77.287,401.881,165.741,53.050,159.493
C04583=1018.837,-77.537,401.891,165.738,53.054,159.493
C04584=1018.830,-77.787,401.901,165.735,53.060,159.493
C04585=1018.826,-78.036,401.910,165.731,53.064,159.493
C04586=1018.820,-78.286,401.921,165.729,53.069,159.494
C04587=1018.815,-78.536,401.931,165.726,53.074,159.494
C04588=1018.809,-78.785,401.940,165.723,53.080,159.494
C04589=1018.804,-79.035,401.950,165.719,53.084,159.495
C04590=1018.799,-79.285,401.960,165.717,53.089,159.495
C04591=1018.793,-79.535,401.969,165.714,53.094,159.495
C04592=1018.787,-79.785,401.980,165.711,53.099,159.496
C04593=1018.782,-80.034,401.989,165.707,53.104,159.496
C04594=1018.777,-80.284,402.000,165.705,53.108,159.496
C04595=1018.771,-80.533,402.009,165.702,53.114,159.496
C04596=1018.766,-80.783,402.019,165.699,53.119,159.497
C04597=1018.761,-81.033,402.027,165.695,53.124,159.497
C04598=1018.755,-81.283,402.038,165.692,53.129,159.497
C04599=1018.750,-81.532,402.047,165.689,53.135,159.497
C04600=1018.743,-81.782,402.056,165.687,53.139,159.498
C04601=1018.738,-82.033,402.066,165.684,53.145,159.498
C04602=1018.733,-82.282,402.075,165.681,53.150,159.498
C04603=1018.727,-82.532,402.085,165.677,53.155,159.499
C04604=1018.722,-82.781,402.094,165.674,53.160,159.499
C04605=1018.717,-83.032,402.104,165.671,53.166,159.499
C04606=1018.711,-83.281,402.113,165.668,53.170,159.499
C04607=1018.706,-83.531,402.123,165.666,53.175,159.500
C04608=1018.700,-83.780,402.132,165.662,53.180,159.500
C04609=1018.695,-84.031,402.142,165.659,53.186,159.500
C04610=1018.689,-84.280,402.151,165.656,53.191,159.501
C04611=1018.684,-84.529,402.160,165.653,53.196,159.501
C04612=1018.679,-84.780,402.170,165.650,53.201,159.501
C04613=1018.673,-85.029,402.179,165.647,53.205,159.501
C04614=1018.667,-85.311,402.190,165.644,53.212,159.502
C04615=1018.661,-85.592,402.201,165.641,53.217,159.502
C04616=1018.654,-85.873,402.211,165.637,53.223,159.502
C04617=1018.649,-86.156,402.221,165.634,53.229,159.503
C04618=1018.643,-86.405,402.231,165.631,53.234,159.503
C04619=1018.638,-86.655,402.241,165.627,53.239,159.503
C04620=1018.633,-86.904,402.249,165.624,53.244,159.504
C04621=1018.628,-87.154,402.259,165.622,53.249,159.504
C04622=1018.622,-87.404,402.269,165.619,53.254,159.504
C04623=1018.617,-87.654,402.278,165.615,53.259,159.504
C04624=1018.611,-87.904,402.287,165.612,53.264,159.505
C04625=1018.606,-88.153,402.296,165.609,53.269,159.505
C04626=1018.601,-88.403,402.305,165.607,53.274,159.505
C04627=1018.595,-88.653,402.314,165.603,53.279,159.505
C04628=1018.590,-88.902,402.324,165.600,53.284,159.506
C04629=1018.584,-89.152,402.334,165.597,53.289,159.506
C04630=1018.579,-89.402,402.343,165.594,53.294,159.506
C04631=1018.574,-89.651,402.352,165.591,53.299,159.507
C04632=1018.568,-89.902,402.361,165.588,53.304,159.507
C04633=1018.563,-90.151,402.371,165.585,53.309,159.507
C04634=1018.558,-90.401,402.379,165.582,53.314,159.507
C04635=1018.552,-90.651,402.389,165.578,53.319,159.507
C04636=1018.547,-90.901,402.398,165.576,53.324,159.508
C04637=1018.542,-91.150,402.408,165.573,53.329,159.508
C04638=1018.536,-91.401,402.416,165.570,53.334,159.508
C04639=1018.531,-91.650,402.426,165.566,53.339,159.509
C04640=1018.526,-91.900,402.435,165.563,53.344,159.509
C04641=1018.521,-92.149,402.443,165.561,53.349,159.509
C04642=1018.516,-92.400,402.453,165.558,53.354,159.510
C04643=1018.510,-92.649,402.462,165.555,53.359,159.510
C04644=1018.505,-92.898,402.471,165.552,53.364,159.510
C04645=1018.500,-93.149,402.480,165.549,53.369,159.510
C04646=1018.494,-93.398,402.490,165.546,53.374,159.511
C04647=1018.490,-93.648,402.499,165.543,53.379,159.511
C04648=1018.484,-93.898,402.507,165.539,53.384,159.511
C04649=1018.479,-94.148,402.517,165.537,53.389,159.511
C04650=1018.474,-94.398,402.526,165.534,53.394,159.511
C04651=1018.468,-94.647,402.535,165.531,53.399,159.512
C04652=1018.463,-94.897,402.544,165.527,53.404,159.512
C04653=1018.458,-95.147,402.553,165.525,53.408,159.512
C04654=1018.453,-95.397,402.563,165.522,53.414,159.513
C04655=1018.448,-95.646,402.571,165.519,53.418,159.513
C04656=1018.442,-95.896,402.580,165.516,53.424,159.513
C04657=1018.437,-96.146,402.590,165.513,53.428,159.513
C04658=1018.432,-96.396,402.598,165.510,53.433,159.513
C04659=1018.427,-96.646,402.607,165.507,53.438,159.514
C04660=1018.421,-96.895,402.617,165.503,53.443,159.514
C04661=1018.416,-97.145,402.625,165.501,53.448,159.514
C04662=1018.412,-97.395,402.634,165.498,53.453,159.514
C04663=1018.406,-97.645,402.643,165.494,53.458,159.515
C04664=1018.401,-97.895,402.653,165.491,53.463,159.515
C04665=1018.396,-98.144,402.661,165.488,53.468,159.515
C04666=1018.390,-98.394,402.670,165.486,53.473,159.515
C04667=1018.385,-98.644,402.678,165.482,53.478,159.516
C04668=1018.380,-98.893,402.687,165.479,53.483,159.516
C04669=1018.374,-99.144,402.696,165.476,53.488,159.516
C04670=1018.369,-99.394,402.704,165.473,53.493,159.516
C04671=1018.363,-99.643,402.713,165.470,53.499,159.517
C04672=1018.359,-99.893,402.722,165.468,53.503,159.517
C04673=1018.353,-100.142,402.731,165.465,53.509,159.517
C04674=1018.348,-100.392,402.739,165.461,53.513,159.517
C04675=1018.343,-100.642,402.748,165.458,53.519,159.518
C04676=1018.338,-100.892,402.756,165.455,53.524,159.518
C04677=1018.332,-101.142,402.765,165.452,53.529,159.518
C04678=1018.327,-101.398,402.774,165.449,53.534,159.518
C04679=1018.322,-101.654,402.783,165.446,53.539,159.519
C04680=1018.316,-101.911,402.791,165.443,53.545,159.519
C04681=1018.311,-102.167,402.800,165.440,53.549,159.519
C04682=1018.306,-102.417,402.809,165.437,53.555,159.520
C04683=1018.300,-102.667,402.817,165.433,53.559,159.520
C04684=1018.295,-102.916,402.826,165.430,53.565,159.520
C04685=1018.291,-103.166,402.835,165.427,53.570,159.520
C04686=1018.285,-103.417,402.843,165.425,53.575,159.521
C04687=1018.279,-103.667,402.852,165.422,53.580,159.521
C04688=1018.274,-103.916,402.860,165.419,53.585,159.521
C04689=1018.269,-104.166,402.869,165.415,53.590,159.521
C04690=1018.264,-104.416,402.877,165.412,53.595,159.522
///RCONF 1,0,0,0,1,0,0,0,0,0,0,0,0,0,0,0,0,0,0,0,0,0,0,0
C04691=1018.258,-104.665,402.886,165.410,53.600,159.522
C04692=1018.253,-104.915,402.894,165.406,53.604,159.522
C04693=1018.248,-105.165,402.903,165.403,53.610,159.522
C04694=1018.242,-105.442,402.913,165.400,53.615,159.523
C04695=1018.237,-105.719,402.922,165.396,53.621,159.523
C04696=1018.231,-105.996,402.931,165.393,53.627,159.523
C04697=1018.225,-106.273,402.940,165.390,53.632,159.523
C04698=1018.219,-106.522,402.949,165.387,53.637,159.524
C04699=1018.215,-106.773,402.957,165.384,53.642,159.524
C04700=1018.209,-107.022,402.965,165.380,53.647,159.524
C04701=1018.204,-107.272,402.974,165.379,53.652,159.524
C04702=1018.199,-107.522,402.983,165.375,53.657,159.525
C04703=1018.194,-107.772,402.991,165.372,53.663,159.525
C04704=1018.189,-108.022,402.999,165.369,53.667,159.525
C04705=1018.183,-108.271,403.007,165.366,53.673,159.525
C04706=1018.179,-108.520,403.015,165.362,53.678,159.525
C04707=1018.173,-108.770,403.023,165.360,53.683,159.526
C04708=1018.168,-109.021,403.031,165.357,53.688,159.526
C04709=1018.163,-109.270,403.040,165.354,53.693,159.526
C04710=1018.158,-109.520,403.048,165.350,53.698,159.526
C04711=1018.153,-109.770,403.057,165.347,53.703,159.527
C04712=1018.148,-110.020,403.064,165.344,53.708,159.527
C04713=1018.142,-110.270,403.073,165.342,53.713,159.527
C04714=1018.136,-110.519,403.081,165.339,53.718,159.528
C04715=1018.131,-110.769,403.089,165.336,53.723,159.528
C04716=1018.126,-111.019,403.097,165.332,53.728,159.528
C04717=1018.121,-111.268,403.105,165.329,53.734,159.528
C04718=1018.116,-111.519,403.113,165.326,53.738,159.528
C04719=1018.111,-111.768,403.121,165.324,53.744,159.529
C04720=1018.106,-112.019,403.129,165.320,53.748,159.529
C04721=1018.101,-112.268,403.138,165.317,53.754,159.529
C04722=1018.096,-112.518,403.146,165.314,53.759,159.529
C04723=1018.090,-112.768,403.153,165.311,53.764,159.530
C04724=1018.085,-113.017,403.162,165.309,53.769,159.530
C04725=1018.080,-113.267,403.169,165.306,53.774,159.530
C04726=1018.075,-113.517,403.178,165.302,53.779,159.530
C04727=1018.070,-113.767,403.186,165.299,53.784,159.531
C04728=1018.065,-114.017,403.194,165.296,53.789,159.531
C04729=1018.060,-114.266,403.202,165.294,53.794,159.531
C04730=1018.055,-114.517,403.210,165.291,53.799,159.531
C04731=1018.049,-114.766,403.218,165.287,53.804,159.532
C04732=1018.044,-115.016,403.226,165.284,53.809,159.532
C04733=1018.039,-115.266,403.234,165.281,53.815,159.532
C04734=1018.035,-115.516,403.241,165.279,53.819,159.532
C04735=1018.029,-115.765,403.250,165.276,53.825,159.533
C04736=1018.024,-116.015,403.257,165.272,53.829,159.533
C04737=1018.018,-116.265,403.266,165.269,53.835,159.533
C04738=1018.014,-116.515,403.273,165.266,53.840,159.533
C04739=1018.009,-116.765,403.281,165.263,53.845,159.534
C04740=1018.003,-117.014,403.289,165.261,53.850,159.534
C04741=1017.998,-117.265,403.296,165.258,53.855,159.534
C04742=1017.993,-117.548,403.306,165.254,53.861,159.534
C04743=1017.986,-117.831,403.315,165.251,53.867,159.535
C04744=1017.981,-118.115,403.323,165.247,53.872,159.535
C04745=1017.975,-118.399,403.332,165.244,53.878,159.535
C04746=1017.970,-118.649,403.340,165.240,53.883,159.535
C04747=1017.965,-118.898,403.347,165.237,53.888,159.536
C04748=1017.960,-119.148,403.355,165.235,53.893,159.536
C04749=1017.955,-119.398,403.363,165.232,53.898,159.536
C04750=1017.950,-119.647,403.371,165.228,53.903,159.536
C04751=1017.944,-119.897,403.378,165.226,53.909,159.537
C04752=1017.939,-120.148,403.386,165.222,53.913,159.537
C04753=1017.935,-120.397,403.394,165.219,53.919,159.537
C04754=1017.929,-120.647,403.401,165.217,53.923,159.537
C04755=1017.924,-120.897,403.409,165.214,53.929,159.538
C04756=1017.920,-121.147,403.416,165.210,53.934,159.538
C04757=1017.914,-121.396,403.424,165.207,53.939,159.538
C04758=1017.909,-121.647,403.432,165.204,53.944,159.538
C04759=1017.904,-121.896,403.439,165.202,53.949,159.539
C04760=1017.899,-122.146,403.447,165.199,53.954,159.539
C04761=1017.893,-122.396,403.455,165.196,53.959,159.539
C04762=1017.889,-122.646,403.462,165.192,53.964,159.539
C04763=1017.883,-122.896,403.470,165.190,53.969,159.540
C04764=1017.879,-123.145,403.477,165.187,53.974,159.540
C04765=1017.874,-123.396,403.485,165.184,53.980,159.540
C04766=1017.868,-123.645,403.493,165.181,53.984,159.540
C04767=1017.864,-123.895,403.500,165.177,53.989,159.540
C04768=1017.859,-124.145,403.508,165.175,53.994,159.541
C04769=1017.854,-124.394,403.515,165.172,53.999,159.541
C04770=1017.849,-124.645,403.522,165.169,54.005,159.541
C04771=1017.843,-124.895,403.530,165.165,54.009,159.541
C04772=1017.839,-125.144,403.537,165.162,54.015,159.542
C04773=1017.833,-125.394,403.544,165.160,54.019,159.542
C04774=1017.829,-125.644,403.552,165.157,54.025,159.542
C04775=1017.823,-125.893,403.559,165.154,54.030,159.542
C04776=1017.818,-126.143,403.567,165.151,54.035,159.542
C04777=1017.813,-126.393,403.574,165.147,54.040,159.543
C04778=1017.808,-126.643,403.581,165.144,54.046,159.543
C04779=1017.803,-126.893,403.589,165.142,54.050,159.543
C04780=1017.798,-127.142,403.596,165.139,54.056,159.543
C04781=1017.792,-127.392,403.603,165.136,54.060,159.544
C04782=1017.788,-127.642,403.611,165.133,54.066,159.544
C04783=1017.782,-127.892,403.618,165.129,54.071,159.544
C04784=1017.778,-128.142,403.625,165.127,54.076,159.544
C04785=1017.774,-128.391,403.633,165.124,54.081,159.545
C04786=1017.770,-128.640,403.641,165.121,54.084,159.545
C04787=1017.765,-128.891,403.650,165.118,54.088,159.545
C04788=1017.762,-129.140,403.660,165.116,54.091,159.545
C04789=1017.759,-129.389,403.670,165.113,54.093,159.544
C04790=1017.757,-129.639,403.681,165.111,54.094,159.544
C04791=1017.755,-129.888,403.692,165.108,54.096,159.544
C04792=1017.752,-130.138,403.705,165.106,54.097,159.543
C04793=1017.751,-130.388,403.717,165.103,54.097,159.543
C04794=1017.751,-130.638,403.731,165.101,54.097,159.542
C04795=1017.750,-130.887,403.744,165.099,54.096,159.542
C04796=1017.750,-131.138,403.759,165.096,54.094,159.541
C04797=1017.751,-131.387,403.774,165.094,54.092,159.540
C04798=1017.751,-131.637,403.789,165.092,54.090,159.539
C04799=1017.753,-131.887,403.806,165.090,54.086,159.538
C04800=1017.754,-132.137,403.822,165.088,54.083,159.537
C04801=1017.756,-132.385,403.839,165.086,54.079,159.536
C04802=1017.759,-132.635,403.857,165.085,54.074,159.535
C04803=1017.762,-132.886,403.875,165.083,54.069,159.533
C04804=1017.765,-133.135,403.894,165.082,54.063,159.532
C04805=1017.769,-133.384,403.915,165.080,54.056,159.531
C04806=1017.507,-133.410,403.534,165.038,54.403,159.582
C04807=1017.503,-133.162,403.514,165.040,54.409,159.583
C04808=1017.500,-132.912,403.495,165.042,54.415,159.585
C04809=1017.497,-132.662,403.476,165.043,54.420,159.586
C04810=1017.495,-132.412,403.458,165.045,54.425,159.587
C04811=1017.493,-132.162,403.441,165.047,54.429,159.588
C04812=1017.491,-131.913,403.424,165.049,54.433,159.589
C04813=1017.490,-131.663,403.409,165.050,54.436,159.590
C04814=1017.489,-131.413,403.393,165.053,54.439,159.591
C04815=1017.488,-131.164,403.378,165.055,54.441,159.592
C04816=1017.489,-130.914,403.364,165.057,54.442,159.593
C04817=1017.489,-130.664,403.350,165.060,54.443,159.594
C04818=1017.490,-130.414,403.336,165.062,54.443,159.594
C04819=1017.491,-130.164,403.323,165.064,54.443,159.594
C04820=1017.493,-129.915,403.312,165.066,54.442,159.595
C04821=1017.495,-129.665,403.300,165.069,54.441,159.595
C04822=1017.497,-129.416,403.290,165.072,54.439,159.596
C04823=1017.500,-129.166,403.279,165.074,54.437,159.596
C04824=1017.504,-128.916,403.269,165.078,54.434,159.596
C04825=1017.508,-128.667,403.261,165.079,54.430,159.596
C04826=1017.512,-128.417,403.252,165.083,54.426,159.596
C04827=1017.516,-128.168,403.244,165.086,54.422,159.596
C04828=1017.521,-127.919,403.236,165.089,54.416,159.595
C04829=1017.526,-127.669,403.229,165.092,54.411,159.595
C04830=1017.531,-127.419,403.222,165.095,54.406,159.595
C04831=1017.536,-127.170,403.215,165.097,54.401,159.595
C04832=1017.541,-126.919,403.207,165.100,54.396,159.594
C04833=1017.546,-126.670,403.200,165.103,54.390,159.594
C04834=1017.551,-126.420,403.193,165.106,54.385,159.594
C04835=1017.556,-126.170,403.186,165.109,54.380,159.594
C04836=1017.561,-125.920,403.178,165.113,54.375,159.593
C04837=1017.566,-125.671,403.171,165.116,54.369,159.593
C04838=1017.571,-125.420,403.163,165.118,54.364,159.593
C04839=1017.577,-125.170,403.156,165.122,54.359,159.593
C04840=1017.581,-124.921,403.149,165.124,54.354,159.592
C04841=1017.587,-124.671,403.142,165.127,54.348,159.592
C04842=1017.591,-124.421,403.134,165.130,54.343,159.592
C04843=1017.596,-124.171,403.127,165.133,54.338,159.592
C04844=1017.601,-123.921,403.120,165.136,54.333,159.591
C04845=1017.606,-123.671,403.112,165.139,54.327,159.591
C04846=1017.611,-123.422,403.105,165.143,54.323,159.591
C04847=1017.616,-123.172,403.097,165.145,54.317,159.591
C04848=1017.621,-122.922,403.089,165.148,54.313,159.590
C04849=1017.626,-122.672,403.082,165.151,54.307,159.590
C04850=1017.631,-122.422,403.074,165.154,54.302,159.590
C04851=1017.636,-122.172,403.067,165.157,54.297,159.590
C04852=1017.641,-121.922,403.060,165.160,54.291,159.589
C04853=1017.647,-121.673,403.051,165.163,54.286,159.589
C04854=1017.651,-121.423,403.044,165.165,54.281,159.589
C04855=1017.657,-121.173,403.037,165.169,54.276,159.589
C04856=1017.661,-120.923,403.029,165.172,54.271,159.588
C04857=1017.666,-120.674,403.021,165.175,54.266,159.588
C04858=1017.672,-120.424,403.014,165.178,54.260,159.588
C04859=1017.676,-120.174,403.006,165.181,54.255,159.588
C04860=1017.681,-119.924,402.998,165.184,54.250,159.588
C04861=1017.687,-119.674,402.990,165.187,54.244,159.587
C04862=1017.692,-119.425,402.983,165.190,54.240,159.587
C04863=1017.697,-119.174,402.975,165.192,54.234,159.587
C04864=1017.702,-118.924,402.968,165.196,54.230,159.586
C04865=1017.707,-118.675,402.960,165.199,54.224,159.586
C04866=1017.712,-118.425,402.952,165.202,54.218,159.586
C04867=1017.718,-118.142,402.944,165.206,54.213,159.586
C04868=1017.723,-117.858,402.935,165.209,54.207,159.585
C04869=1017.730,-117.575,402.926,165.213,54.201,159.585
C04870=1017.735,-117.291,402.917,165.215,54.195,159.585
C04871=1017.740,-117.041,402.909,165.218,54.190,159.585
C04872=1017.746,-116.792,402.902,165.221,54.184,159.584
C04873=1017.751,-116.542,402.894,165.225,54.180,159.584
C04874=1017.755,-116.291,402.886,165.228,54.174,159.584
C04875=1017.760,-116.042,402.878,165.231,54.169,159.584
C04876=1017.766,-115.792,402.871,165.234,54.164,159.583
C04877=1017.771,-115.542,402.862,165.236,54.159,159.583
C04878=1017.776,-115.292,402.854,165.239,54.154,159.583
C04879=1017.781,-115.043,402.846,165.242,54.148,159.582
C04880=1017.786,-114.793,402.839,165.245,54.143,159.582
C04881=1017.791,-114.543,402.831,165.249,54.138,159.582
C04882=1017.797,-114.293,402.823,165.252,54.132,159.582
C04883=1017.801,-114.044,402.815,165.255,54.128,159.582
C04884=1017.806,-113.794,402.807,165.258,54.122,159.581
C04885=1017.812,-113.544,402.799,165.260,54.118,159.581
C04886=1017.816,-113.294,402.791,165.263,54.112,159.581
C04887=1017.822,-113.044,402.782,165.267,54.107,159.581
C04888=1017.827,-112.795,402.775,165.270,54.102,159.580
C04889=1017.832,-112.545,402.767,165.272,54.096,159.580
C04890=1017.837,-112.295,402.759,165.276,54.091,159.580
C04891=1017.842,-112.045,402.751,165.279,54.086,159.579
C04892=1017.848,-111.795,402.742,165.282,54.081,159.579
C04893=1017.852,-111.545,402.735,165.285,54.075,159.579
C04894=1017.857,-111.296,402.726,165.287,54.070,159.579
C04895=1017.862,-111.045,402.719,165.290,54.066,159.578
C04896=1017.868,-110.796,402.711,165.293,54.060,159.578
C04897=1017.873,-110.546,402.702,165.297,54.055,159.578
C04898=1017.878,-110.296,402.694,165.300,54.050,159.578
C04899=1017.884,-110.046,402.686,165.303,54.044,159.577
C04900=1017.888,-109.797,402.678,165.306,54.039,159.577
C04901=1017.893,-109.547,402.670,165.309,54.034,159.577
C04902=1017.899,-109.297,402.662,165.312,54.028,159.577
C04903=1017.904,-109.047,402.653,165.315,54.023,159.576
C04904=1017.909,-108.797,402.645,165.317,54.018,159.576
C04905=1017.914,-108.547,402.637,165.321,54.014,159.576
C04906=1017.920,-108.298,402.629,165.324,54.008,159.576
C04907=1017.925,-108.048,402.621,165.327,54.002,159.575
C04908=1017.930,-107.798,402.613,165.330,53.998,159.575
C04909=1017.936,-107.548,402.604,165.333,53.992,159.575
C04910=1017.941,-107.299,402.596,165.336,53.987,159.574
C04911=1017.945,-107.049,402.588,165.339,53.982,159.574
C04912=1017.950,-106.799,402.580,165.342,53.976,159.574
C04913=1017.956,-106.549,402.571,165.346,53.972,159.574
C04914=1017.961,-106.300,402.563,165.348,53.966,159.573
C04915=1017.965,-106.050,402.554,165.351,53.962,159.573
C04916=1017.971,-105.800,402.545,165.354,53.956,159.573
C04917=1017.976,-105.550,402.538,165.357,53.951,159.573
C04918=1017.981,-105.300,402.529,165.360,53.946,159.572
C04919=1017.986,-105.050,402.521,165.363,53.940,159.572
C04920=1017.991,-104.801,402.512,165.367,53.935,159.572
C04921=1017.997,-104.551,402.504,165.370,53.930,159.572
C04922=1018.002,-104.301,402.495,165.372,53.926,159.571
C04923=1018.007,-104.051,402.487,165.375,53.920,159.571
C04924=1018.013,-103.802,402.478,165.378,53.915,159.571
C04925=1018.018,-103.552,402.470,165.381,53.910,159.571
C04926=1018.023,-103.302,402.461,165.384,53.904,159.570
C04927=1018.027,-103.052,402.453,165.388,53.899,159.570
///RCONF 1,0,0,0,0,0,0,0,0,0,0,0,0,0,0,0,0,0,0,0,0,0,0,0
C04928=1018.033,-102.802,402.444,165.391,53.894,159.570
C04929=1018.038,-102.552,402.436,165.393,53.888,159.570
C04930=1018.043,-102.302,402.427,165.396,53.884,159.569
C04931=1018.049,-102.019,402.417,165.400,53.878,159.569
C04932=1018.055,-101.735,402.408,165.403,53.872,159.569
C04933=1018.061,-101.452,402.398,165.406,53.866,159.568
C04934=1018.068,-101.169,402.388,165.410,53.860,159.568
C04935=1018.072,-100.919,402.379,165.413,53.855,159.568
C04936=1018.077,-100.669,402.371,165.417,53.850,159.568
C04937=1018.083,-100.419,402.362,165.419,53.845,159.567
C04938=1018.088,-100.169,402.354,165.422,53.839,159.567
C04939=1018.093,-99.920,402.345,165.425,53.834,159.567
C04940=1018.099,-99.670,402.337,165.428,53.829,159.566
C04941=1018.104,-99.420,402.328,165.431,53.823,159.566
C04942=1018.109,-99.171,402.320,165.434,53.819,159.566
C04943=1018.115,-98.922,402.311,165.437,53.813,159.566
C04944=1018.120,-98.671,402.301,165.440,53.808,159.565
C04945=1018.125,-98.421,402.293,165.444,53.803,159.565
C04946=1018.130,-98.171,402.284,165.447,53.797,159.565
C04947=1018.136,-97.922,402.276,165.450,53.792,159.564
C04948=1018.141,-97.672,402.267,165.452,53.787,159.564
C04949=1018.145,-97.422,402.258,165.455,53.782,159.564
C04950=1018.151,-97.172,402.249,165.458,53.777,159.564
C04951=1018.156,-96.922,402.240,165.461,53.772,159.563
C04952=1018.161,-96.672,402.231,165.465,53.767,159.563
C04953=1018.167,-96.423,402.223,165.468,53.761,159.563
C04954=1018.171,-96.173,402.213,165.470,53.757,159.563
C04955=1018.177,-95.924,402.204,165.473,53.752,159.562
C04956=1018.182,-95.673,402.195,165.476,53.747,159.562
C04957=1018.187,-95.424,402.186,165.479,53.741,159.562
C04958=1018.193,-95.174,402.177,165.483,53.737,159.562
C04959=1018.197,-94.924,402.168,165.485,53.731,159.561
C04960=1018.203,-94.675,402.159,165.488,53.727,159.561
C04961=1018.207,-94.425,402.150,165.491,53.721,159.561
C04962=1018.213,-94.174,402.141,165.495,53.716,159.561
C04963=1018.219,-93.925,402.132,165.498,53.711,159.560
C04964=1018.223,-93.675,402.123,165.501,53.706,159.560
C04965=1018.228,-93.426,402.114,165.504,53.701,159.560
C04966=1018.234,-93.175,402.104,165.506,53.696,159.560
C04967=1018.243,-92.766,402.090,165.511,53.687,159.559
C04968=1018.251,-92.356,402.075,165.516,53.679,159.559
C04969=1018.260,-91.947,402.060,165.521,53.671,159.558
C04970=1018.268,-91.537,402.045,165.526,53.663,159.558
C04971=1018.274,-91.288,402.036,165.529,53.657,159.557
C04972=1018.279,-91.038,402.026,165.533,53.652,159.557
C04973=1018.284,-90.789,402.017,165.536,53.647,159.557
C04974=1018.289,-90.539,402.008,165.539,53.641,159.557
C04975=1018.294,-90.289,402.000,165.542,53.637,159.557
C04976=1018.300,-90.039,401.989,165.544,53.631,159.556
C04977=1018.305,-89.789,401.981,165.547,53.627,159.556
C04978=1018.310,-89.540,401.972,165.550,53.621,159.556
C04979=1018.316,-89.289,401.962,165.553,53.616,159.555
C04980=1018.321,-89.040,401.953,165.557,53.611,159.555
C04981=1018.326,-88.790,401.944,165.560,53.606,159.555
C04982=1018.332,-88.540,401.934,165.563,53.600,159.554
C04983=1018.336,-88.290,401.925,165.566,53.595,159.554
C04984=1018.342,-88.041,401.916,165.568,53.590,159.554
C04985=1018.348,-87.791,401.907,165.571,53.585,159.553
C04986=1018.353,-87.541,401.898,165.575,53.580,159.553
C04987=1018.359,-87.292,401.888,165.577,53.575,159.553
C04988=1018.363,-87.041,401.879,165.580,53.569,159.553
C04989=1018.369,-86.792,401.870,165.584,53.564,159.553
C04990=1018.374,-86.542,401.860,165.587,53.559,159.552
C04991=1018.383,-86.171,401.846,165.591,53.551,159.552
C04992=1018.390,-85.799,401.833,165.595,53.543,159.551
C04993=1018.398,-85.428,401.819,165.600,53.535,159.551
C04994=1018.406,-85.057,401.805,165.605,53.528,159.550
C04995=1018.412,-84.807,401.795,165.608,53.523,159.550
C04996=1018.417,-84.557,401.786,165.611,53.518,159.550
C04997=1018.423,-84.308,401.777,165.614,53.512,159.550
C04998=1018.428,-84.058,401.767,165.617,53.507,159.549
C04999=1018.434,-83.808,401.758,165.620,53.502,159.549
C05000=1018.438,-83.558,401.748,165.623,53.496,159.549
C05001=1018.445,-83.309,401.739,165.625,53.491,159.548
C05002=1018.449,-83.059,401.730,165.628,53.486,159.548
C05003=1018.455,-82.809,401.720,165.632,53.481,159.548
C05004=1018.461,-82.560,401.711,165.635,53.476,159.547
C05005=1018.465,-82.310,401.702,165.638,53.470,159.547
C05006=1018.472,-82.060,401.692,165.641,53.465,159.547
C05007=1018.476,-81.810,401.682,165.644,53.460,159.547
C05008=1018.483,-81.561,401.673,165.647,53.455,159.546
C05009=1018.487,-81.311,401.664,165.650,53.449,159.546
C05010=1018.493,-81.061,401.654,165.653,53.444,159.545
C05011=1018.498,-80.811,401.644,165.657,53.439,159.545
C05012=1018.504,-80.562,401.635,165.660,53.433,159.545
C05013=1018.509,-80.311,401.625,165.663,53.428,159.545
C05014=1018.515,-80.062,401.616,165.666,53.423,159.544
C05015=1018.520,-79.812,401.606,165.668,53.418,159.544
C05016=1018.525,-79.562,401.596,165.671,53.413,159.544
C05017=1018.531,-79.312,401.587,165.674,53.408,159.544
C05018=1018.536,-79.063,401.577,165.677,53.403,159.543
C05019=1018.542,-78.813,401.567,165.680,53.397,159.543
C05020=1018.546,-78.564,401.557,165.684,53.392,159.543
C05021=1018.553,-78.314,401.547,165.686,53.387,159.542
C05022=1018.558,-78.064,401.537,165.689,53.383,159.542
C05023=1018.563,-77.814,401.527,165.692,53.377,159.542
C05024=1018.569,-77.564,401.518,165.695,53.372,159.541
C05025=1018.574,-77.315,401.508,165.699,53.367,159.541
C05026=1018.579,-77.065,401.498,165.702,53.361,159.541
C05027=1018.584,-76.815,401.488,165.704,53.356,159.540
C05028=1018.590,-76.566,401.478,165.707,53.352,159.540
C05029=1018.596,-76.316,401.468,165.710,53.346,159.540
C05030=1018.601,-76.066,401.458,165.713,53.341,159.540
C05031=1018.606,-75.816,401.448,165.717,53.336,159.539
C05032=1018.612,-75.566,401.439,165.719,53.331,159.539
C05033=1018.617,-75.317,401.429,165.722,53.325,159.539
C05034=1018.622,-75.067,401.419,165.726,53.320,159.539
C05035=1018.627,-74.817,401.409,165.728,53.315,159.538
C05036=1018.633,-74.568,401.399,165.731,53.310,159.538
C05037=1018.639,-74.317,401.389,165.734,53.305,159.538
C05038=1018.644,-74.068,401.379,165.737,53.300,159.537
C05039=1018.649,-73.819,401.369,165.741,53.295,159.537
C05040=1018.655,-73.568,401.358,165.743,53.290,159.537
C05041=1018.660,-73.319,401.349,165.746,53.285,159.536
C05042=1018.665,-73.069,401.338,165.749,53.280,159.536
C05043=1018.671,-72.819,401.328,165.753,53.275,159.536
C05044=1018.675,-72.570,401.317,165.755,53.270,159.535
C05045=1018.680,-72.320,401.307,165.758,53.265,159.535
C05046=1018.686,-72.069,401.297,165.761,53.260,159.535
C05047=1018.691,-71.821,401.286,165.765,53.255,159.535
C05048=1018.696,-71.571,401.276,165.766,53.250,159.534
C05049=1018.702,-71.320,401.266,165.770,53.245,159.534
C05050=1018.708,-71.071,401.255,165.773,53.240,159.534
C05051=1018.712,-70.822,401.245,165.776,53.235,159.534
C05052=1018.718,-70.571,401.235,165.778,53.230,159.533
C05053=1018.723,-70.321,401.225,165.782,53.225,159.533
C05054=1018.728,-70.073,401.215,165.785,53.220,159.533
C05055=1018.734,-69.793,401.203,165.788,53.215,159.532
C05056=1018.741,-69.513,401.192,165.792,53.209,159.532
C05057=1018.746,-69.234,401.180,165.795,53.203,159.532
C05058=1018.752,-68.955,401.168,165.798,53.198,159.531
C05059=1018.758,-68.705,401.157,165.801,53.192,159.531
C05060=1018.763,-68.455,401.147,165.804,53.188,159.531
C05061=1018.768,-68.206,401.137,165.807,53.182,159.530
C05062=1018.774,-67.956,401.126,165.810,53.178,159.530
C05063=1018.779,-67.706,401.116,165.813,53.173,159.530
C05064=1018.785,-67.456,401.105,165.816,53.167,159.529
C05065=1018.791,-67.206,401.095,165.819,53.162,159.529
C05066=1018.795,-66.957,401.085,165.822,53.157,159.529
C05067=1018.801,-66.707,401.075,165.825,53.153,159.529
C05068=1018.807,-66.457,401.064,165.828,53.147,159.528
C05069=1018.812,-66.208,401.054,165.831,53.142,159.528
C05070=1018.818,-65.958,401.043,165.834,53.137,159.528
C05071=1018.823,-65.709,401.033,165.837,53.132,159.527
C05072=1018.828,-65.459,401.023,165.839,53.127,159.527
C05073=1018.834,-65.209,401.012,165.843,53.122,159.527
C05074=1018.839,-64.959,401.001,165.846,53.116,159.526
C05075=1018.845,-64.709,400.990,165.849,53.112,159.526
C05076=1018.850,-64.459,400.980,165.852,53.106,159.526
C05077=1018.856,-64.210,400.969,165.854,53.101,159.525
C05078=1018.861,-63.960,400.959,165.858,53.097,159.525
C05079=1018.866,-63.711,400.948,165.861,53.091,159.525
C05080=1018.872,-63.461,400.938,165.864,53.086,159.525
C05081=1018.877,-63.211,400.927,165.867,53.081,159.524
C05082=1018.883,-62.961,400.917,165.869,53.076,159.524
C05083=1018.889,-62.712,400.906,165.872,53.071,159.524
C05084=1018.894,-62.462,400.896,165.875,53.065,159.523
C05085=1018.900,-62.212,400.885,165.879,53.061,159.523
C05086=1018.906,-61.963,400.874,165.882,53.055,159.523
C05087=1018.910,-61.713,400.865,165.885,53.050,159.522
C05088=1018.915,-61.463,400.853,165.887,53.045,159.522
C05089=1018.921,-61.214,400.842,165.890,53.040,159.522
C05090=1018.927,-60.964,400.832,165.893,53.035,159.521
C05091=1018.932,-60.714,400.821,165.896,53.029,159.521
C05092=1018.938,-60.464,400.811,165.900,53.024,159.521
C05093=1018.943,-60.215,400.800,165.903,53.019,159.520
C05094=1018.949,-59.965,400.789,165.905,53.014,159.520
C05095=1018.955,-59.715,400.779,165.908,53.009,159.520
C05096=1018.960,-59.466,400.768,165.911,53.004,159.519
C05097=1018.966,-59.216,400.757,165.914,52.998,159.519
C05098=1018.972,-58.966,400.747,165.917,52.993,159.519
C05099=1018.977,-58.717,400.736,165.920,52.988,159.518
C05100=1018.982,-58.467,400.725,165.923,52.983,159.518
C05101=1018.988,-58.217,400.715,165.926,52.978,159.518
C05102=1018.993,-57.967,400.704,165.929,52.973,159.517
C05103=1018.999,-57.718,400.693,165.932,52.967,159.517
C05104=1019.005,-57.468,400.682,165.935,52.962,159.517
C05105=1019.010,-57.218,400.672,165.938,52.957,159.516
C05106=1019.016,-56.969,400.661,165.941,52.952,159.516
C05107=1019.022,-56.719,400.650,165.943,52.947,159.515
C05108=1019.028,-56.470,400.639,165.946,52.941,159.515
C05109=1019.033,-56.220,400.629,165.949,52.936,159.515
C05110=1019.038,-55.970,400.618,165.953,52.931,159.515
C05111=1019.044,-55.720,400.607,165.956,52.926,159.514
C05112=1019.050,-55.471,400.596,165.959,52.920,159.514
C05113=1019.055,-55.221,400.586,165.962,52.915,159.513
C05114=1019.061,-54.971,400.575,165.964,52.910,159.513
C05115=1019.066,-54.722,400.564,165.967,52.904,159.513
C05116=1019.073,-54.471,400.553,165.970,52.900,159.512
C05117=1019.079,-54.222,400.542,165.973,52.894,159.512
C05118=1019.084,-53.972,400.532,165.976,52.889,159.512
C05119=1019.090,-53.694,400.519,165.979,52.883,159.511
C05120=1019.096,-53.416,400.507,165.983,52.877,159.511
C05121=1019.102,-53.138,400.495,165.986,52.872,159.511
C05122=1019.109,-52.859,400.482,165.990,52.865,159.510
C05123=1019.115,-52.609,400.472,165.992,52.860,159.510
C05124=1019.120,-52.360,400.461,165.995,52.855,159.509
C05125=1019.126,-52.110,400.451,165.998,52.849,159.509
C05126=1019.132,-51.861,400.440,166.001,52.844,159.508
C05127=1019.138,-51.611,400.429,166.004,52.839,159.508
C05128=1019.143,-51.361,400.417,166.007,52.834,159.508
C05129=1019.149,-51.111,400.406,166.010,52.829,159.508
C05130=1019.155,-50.862,400.395,166.013,52.823,159.507
C05131=1019.160,-50.612,400.384,166.015,52.818,159.507
C05132=1019.165,-50.363,400.373,166.019,52.814,159.507
C05133=1019.170,-50.113,400.361,166.022,52.808,159.506
C05134=1019.176,-49.863,400.350,166.024,52.803,159.506
C05135=1019.182,-49.613,400.339,166.027,52.798,159.505
C05136=1019.188,-49.364,400.327,166.030,52.793,159.505
C05137=1019.193,-49.114,400.316,166.033,52.788,159.505
C05138=1019.198,-48.865,400.305,166.036,52.783,159.504
C05139=1019.203,-48.615,400.293,166.039,52.778,159.504
C05140=1019.210,-48.365,400.282,166.042,52.773,159.504
C05141=1019.215,-48.115,400.270,166.045,52.768,159.504
C05142=1019.221,-47.865,400.260,166.047,52.763,159.503
C05143=1019.226,-47.616,400.247,166.050,52.758,159.503
C05144=1019.232,-47.367,400.237,166.054,52.753,159.502
C05145=1019.237,-47.116,400.225,166.057,52.748,159.502
C05146=1019.243,-46.867,400.214,166.059,52.743,159.502
C05147=1019.248,-46.617,400.202,166.063,52.738,159.501
C05148=1019.254,-46.368,400.191,166.066,52.733,159.501
C05149=1019.259,-46.118,400.179,166.068,52.727,159.501
C05150=1019.265,-45.868,400.168,166.071,52.722,159.500
C05151=1019.270,-45.618,400.157,166.074,52.717,159.500
C05152=1019.276,-45.369,400.145,166.077,52.712,159.500
C05153=1019.281,-45.120,400.134,166.080,52.707,159.499
C05154=1019.288,-44.869,400.122,166.082,52.702,159.499
C05155=1019.293,-44.620,400.111,166.086,52.697,159.499
C05156=1019.298,-44.370,400.099,166.089,52.692,159.498
C05157=1019.304,-44.120,400.087,166.092,52.686,159.498
C05158=1019.309,-43.870,400.076,166.094,52.681,159.497
C05159=1019.315,-43.621,400.064,166.097,52.677,159.497
C05160=1019.320,-43.372,400.053,166.100,52.671,159.497
C05161=1019.327,-43.121,400.042,166.103,52.666,159.496
C05162=1019.332,-42.872,400.029,166.105,52.661,159.496
C05163=1019.338,-42.623,400.019,166.108,52.656,159.496
C05164=1019.343,-42.372,400.007,166.112,52.651,159.495
C05165=1019.349,-42.123,399.995,166.115,52.646,159.495
C05166=1019.354,-41.874,399.984,166.117,52.641,159.494
C05167=1019.361,-41.623,399.972,166.120,52.635,159.494
C05168=1019.366,-41.374,399.960,166.123,52.630,159.494
C05169=1019.372,-41.125,399.949,166.127,52.625,159.494
C05170=1019.377,-40.874,399.937,166.130,52.620,159.493
C05171=1019.383,-40.625,399.925,166.132,52.615,159.493
C05172=1019.388,-40.376,399.914,166.135,52.609,159.492
C05173=1019.394,-40.126,399.902,166.138,52.604,159.492
C05174=1019.400,-39.876,399.891,166.141,52.599,159.492
C05175=1019.405,-39.627,399.879,166.143,52.594,159.491
C05176=1019.412,-39.377,399.868,166.146,52.589,159.491
C05177=1019.417,-39.127,399.856,166.149,52.584,159.490
C05178=1019.423,-38.877,399.844,166.153,52.578,159.490
C05179=1019.428,-38.628,399.831,166.155,52.573,159.490
C05180=1019.434,-38.379,399.820,166.158,52.569,159.489
C05181=1019.440,-38.129,399.808,166.161,52.563,159.489
C05182=1019.445,-37.879,399.796,166.163,52.558,159.488
C05183=1019.451,-37.600,399.783,166.167,52.553,159.488
C05184=1019.457,-37.323,399.770,166.170,52.547,159.488
C05185=1019.463,-37.045,399.757,166.173,52.541,159.487
C05186=1019.470,-36.767,399.743,166.176,52.536,159.487
C05187=1019.475,-36.518,399.731,166.179,52.530,159.487
C05188=1019.481,-36.268,399.719,166.183,52.526,159.486
C05189=1019.486,-36.018,399.707,166.185,52.521,159.486
C05190=1019.491,-35.769,399.695,166.188,52.516,159.485
C05191=1019.498,-35.519,399.683,166.191,52.510,159.485
C05192=1019.503,-35.269,399.672,166.194,52.506,159.485
C05193=1019.509,-35.020,399.659,166.196,52.501,159.484
C05194=1019.514,-34.770,399.647,166.199,52.495,159.484
C05195=1019.520,-34.520,399.635,166.202,52.490,159.484
C05196=1019.525,-34.271,399.623,166.204,52.485,159.483
C05197=1019.532,-34.021,399.611,166.208,52.480,159.483
C05198=1019.537,-33.771,399.599,166.211,52.475,159.483
C05199=1019.543,-33.521,399.587,166.214,52.470,159.482
C05200=1019.548,-33.272,399.575,166.216,52.465,159.482
C05201=1019.554,-33.022,399.563,166.219,52.459,159.481
C05202=1019.559,-32.773,399.551,166.222,52.454,159.481
C05203=1019.566,-32.523,399.539,166.226,52.449,159.481
C05204=1019.571,-32.274,399.526,166.228,52.444,159.480
C05205=1019.576,-32.023,399.515,166.231,52.439,159.480
C05206=1019.582,-31.774,399.502,166.234,52.434,159.479
C05207=1019.588,-31.524,399.490,166.237,52.428,159.479
C05208=1019.593,-31.275,399.478,166.239,52.423,159.479
C05209=1019.600,-31.026,399.466,166.242,52.418,159.478
C05210=1019.605,-30.776,399.454,166.245,52.413,159.478
C05211=1019.611,-30.526,399.442,166.247,52.408,159.477
C05212=1019.616,-30.277,399.429,166.251,52.403,159.477
C05213=1019.622,-30.027,399.417,166.254,52.398,159.477
C05214=1019.628,-29.777,399.404,166.257,52.392,159.476
C05215=1019.633,-29.527,399.394,166.260,52.387,159.476
C05216=1019.639,-29.278,399.381,166.262,52.382,159.475
C05217=1019.645,-29.028,399.369,166.265,52.377,159.475
C05218=1019.651,-28.778,399.356,166.268,52.371,159.475
C05219=1019.656,-28.529,399.344,166.271,52.366,159.474
C05220=1019.662,-28.279,399.331,166.273,52.361,159.474
C05221=1019.668,-28.030,399.320,166.276,52.356,159.473
C05222=1019.673,-27.780,399.308,166.279,52.350,159.473
C05223=1019.679,-27.530,399.295,166.282,52.345,159.473
C05224=1019.685,-27.281,399.283,166.284,52.340,159.472
C05225=1019.691,-27.031,399.271,166.288,52.335,159.472
C05226=1019.696,-26.781,399.258,166.291,52.330,159.471
C05227=1019.701,-26.532,399.245,166.293,52.325,159.471
C05228=1019.707,-26.282,399.233,166.296,52.320,159.471
C05229=1019.713,-26.032,399.220,166.299,52.314,159.470
C05230=1019.718,-25.783,399.208,166.302,52.310,159.470
C05231=1019.724,-25.533,399.196,166.305,52.305,159.469
C05232=1019.730,-25.283,399.183,166.308,52.300,159.469
C05233=1019.736,-25.034,399.170,166.310,52.295,159.469
C05234=1019.741,-24.784,399.157,166.313,52.289,159.468
C05235=1019.746,-24.535,399.145,166.316,52.284,159.468
C05236=1019.752,-24.285,399.132,166.318,52.279,159.467
C05237=1019.758,-24.035,399.120,166.322,52.274,159.467
C05238=1019.763,-23.786,399.107,166.325,52.269,159.467
C05239=1019.769,-23.536,399.095,166.327,52.264,159.466
C05240=1019.775,-23.286,399.082,166.330,52.259,159.466
C05241=1019.780,-23.037,399.070,166.333,52.253,159.465
C05242=1019.785,-22.787,399.057,166.335,52.248,159.465
C05243=1019.792,-22.538,399.044,166.338,52.243,159.465
C05244=1019.798,-22.288,399.031,166.341,52.238,159.464
C05245=1019.803,-22.039,399.019,166.344,52.232,159.464
C05246=1019.809,-21.789,399.006,166.347,52.228,159.463
C05247=1019.815,-21.510,398.992,166.351,52.222,159.463
C05248=1019.821,-21.231,398.978,166.353,52.216,159.462
C05249=1019.828,-20.953,398.964,166.356,52.211,159.462
C05250=1019.835,-20.674,398.949,166.359,52.205,159.461
C05251=1019.840,-20.424,398.937,166.362,52.199,159.461
C05252=1019.846,-20.175,398.925,166.366,52.195,159.461
C05253=1019.852,-19.925,398.912,166.368,52.190,159.460
C05254=1019.857,-19.675,398.898,166.371,52.184,159.460
C05255=1019.862,-19.426,398.886,166.374,52.179,159.459
C05256=1019.868,-19.176,398.874,166.377,52.174,159.459
C05257=1019.874,-18.926,398.861,166.379,52.169,159.459
C05258=1019.880,-18.676,398.848,166.382,52.163,159.458
C05259=1019.886,-18.428,398.836,166.385,52.158,159.458
C05260=1019.892,-18.178,398.823,166.387,52.153,159.457
C05261=1019.897,-17.928,398.810,166.390,52.148,159.457
C05262=1019.903,-17.678,398.797,166.393,52.142,159.456
C05263=1019.908,-17.429,398.784,166.396,52.137,159.456
C05264=1019.914,-17.179,398.772,166.398,52.132,159.455
C05265=1019.920,-16.929,398.759,166.401,52.126,159.455
C05266=1019.926,-16.680,398.746,166.404,52.121,159.455
C05267=1019.932,-16.430,398.733,166.407,52.116,159.454
C05268=1019.937,-16.180,398.720,166.410,52.111,159.454
C05269=1019.943,-15.932,398.707,166.413,52.105,159.453
C05270=1019.949,-15.682,398.695,166.416,52.100,159.453
C05271=1019.954,-15.432,398.681,166.418,52.095,159.452
C05272=1019.960,-15.182,398.668,166.421,52.090,159.452
C05273=1019.966,-14.932,398.656,166.424,52.085,159.452
C05274=1019.971,-14.683,398.642,166.426,52.080,159.451
C05275=1019.977,-14.434,398.630,166.430,52.075,159.451
C05276=1019.983,-14.184,398.616,166.433,52.070,159.450
C05277=1019.988,-13.934,398.603,166.435,52.065,159.450
C05278=1019.995,-13.685,398.590,166.438,52.060,159.450
C05279=1020.000,-13.435,398.577,166.441,52.054,159.449
C05280=1020.006,-13.185,398.564,166.443,52.049,159.449
C05281=1020.011,-12.936,398.551,166.446,52.044,159.448
C05282=1020.017,-12.687,398.538,166.449,52.039,159.448
C05283=1020.022,-12.437,398.524,166.451,52.034,159.447
C05284=1020.028,-12.187,398.511,166.454,52.028,159.447
C05285=1020.034,-11.938,398.498,166.458,52.023,159.447
C05286=1020.040,-11.688,398.485,166.460,52.018,159.446
C05287=1020.046,-11.438,398.472,166.463,52.013,159.446
C05288=1020.051,-11.188,398.458,166.466,52.008,159.445
C05289=1020.057,-10.940,398.445,166.468,52.003,159.445
C05290=1020.062,-10.689,398.432,166.471,51.997,159.444
C05291=1020.068,-10.440,398.419,166.474,51.992,159.444
C05292=1020.074,-10.191,398.406,166.476,51.987,159.443
C05293=1020.079,-9.941,398.393,166.479,51.982,159.443
C05294=1020.086,-9.691,398.379,166.482,51.977,159.443
C05295=1020.091,-9.441,398.366,166.485,51.972,159.442
C05296=1020.097,-9.192,398.353,166.488,51.966,159.442
C05297=1020.102,-8.942,398.339,166.491,51.961,159.441
C05298=1020.108,-8.693,398.327,166.493,51.956,159.441
C05299=1020.115,-8.443,398.313,166.496,51.951,159.440
C05300=1020.120,-8.194,398.299,166.499,51.946,159.440
C05301=1020.126,-7.944,398.287,166.501,51.941,159.439
C05302=1020.131,-7.694,398.273,166.504,51.935,159.439
C05303=1020.138,-7.445,398.260,166.507,51.929,159.438
C05304=1020.143,-7.195,398.247,166.510,51.924,159.438
C05305=1020.149,-6.946,398.233,166.512,51.919,159.437
C05306=1020.155,-6.697,398.220,166.515,51.914,159.437
C05307=1020.160,-6.447,398.207,166.518,51.909,159.437
C05308=1020.166,-6.198,398.194,166.520,51.904,159.436
C05309=1020.171,-5.948,398.180,166.524,51.898,159.436
C05310=1020.178,-5.699,398.167,166.527,51.893,159.435
C05311=1020.184,-5.417,398.152,166.529,51.887,159.435
C05312=1020.191,-5.137,398.136,166.532,51.881,159.434
C05313=1020.198,-4.856,398.122,166.536,51.875,159.434
C05314=1020.204,-4.575,398.107,166.539,51.869,159.433
C05315=1020.210,-4.326,398.094,166.542,51.864,159.433
C05316=1020.215,-4.077,398.080,166.544,51.859,159.432
C05317=1020.221,-3.827,398.066,166.547,51.853,159.432
C05318=1020.226,-3.577,398.052,166.549,51.848,159.431
C05319=1020.232,-3.328,398.038,166.552,51.843,159.431
C05320=1020.238,-3.079,398.025,166.555,51.838,159.430
C05321=1020.244,-2.829,398.011,166.557,51.833,159.430
C05322=1020.249,-2.579,397.997,166.561,51.828,159.430
C05323=1020.254,-2.329,397.984,166.563,51.824,159.429
C05324=1020.260,-2.080,397.970,166.566,51.818,159.429
C05325=1020.266,-1.830,397.957,166.569,51.813,159.428
C05326=1020.271,-1.581,397.943,166.571,51.808,159.428
C05327=1020.277,-1.331,397.929,166.574,51.803,159.427
C05328=1020.283,-1.081,397.915,166.577,51.798,159.427
C05329=1020.288,-0.831,397.901,166.580,51.793,159.426
C05330=1020.295,-0.582,397.888,166.583,51.787,159.426
C05331=1020.300,-0.333,397.874,166.585,51.782,159.426
C05332=1020.306,-0.083,397.860,166.588,51.777,159.425
C05333=1020.311,0.167,397.846,166.590,51.772,159.425
C05334=1020.317,0.416,397.832,166.593,51.767,159.424
C05335=1020.322,0.665,397.818,166.596,51.762,159.424
C05336=1020.329,0.914,397.805,166.598,51.756,159.423
C05337=1020.334,1.164,397.791,166.601,51.751,159.423
C05338=1020.339,1.413,397.777,166.603,51.746,159.422
C05339=1020.345,1.663,397.763,166.606,51.741,159.422
C05340=1020.351,1.913,397.749,166.610,51.735,159.421
C05341=1020.357,2.163,397.736,166.612,51.731,159.421
C05342=1020.363,2.412,397.722,166.615,51.725,159.420
C05343=1020.368,2.662,397.708,166.618,51.720,159.420
C05344=1020.374,2.911,397.694,166.620,51.715,159.419
C05345=1020.379,3.161,397.680,166.623,51.710,159.419
C05346=1020.385,3.410,397.666,166.625,51.705,159.419
C05347=1020.392,3.660,397.652,166.628,51.700,159.418
C05348=1020.397,3.909,397.638,166.631,51.694,159.418
C05349=1020.403,4.159,397.624,166.633,51.689,159.417
C05350=1020.408,4.409,397.610,166.636,51.684,159.417
C05351=1020.414,4.658,397.596,166.640,51.678,159.416
C05352=1020.420,4.907,397.583,166.642,51.673,159.416
C05353=1020.426,5.158,397.569,166.645,51.668,159.415
C05354=1020.432,5.407,397.554,166.648,51.663,159.415
C05355=1020.437,5.656,397.540,166.650,51.657,159.414
C05356=1020.443,5.906,397.527,166.653,51.652,159.414
C05357=1020.448,6.155,397.513,166.655,51.647,159.413
C05358=1020.455,6.405,397.499,166.658,51.642,159.413
C05359=1020.461,6.654,397.484,166.661,51.637,159.412
C05360=1020.466,6.904,397.471,166.663,51.631,159.412
C05361=1020.472,7.153,397.457,166.666,51.626,159.411
C05362=1020.477,7.403,397.443,166.669,51.621,159.411
C05363=1020.483,7.653,397.429,166.671,51.616,159.410
C05364=1020.490,7.902,397.415,166.674,51.610,159.410
C05365=1020.495,8.152,397.401,166.677,51.605,159.409
C05366=1020.501,8.401,397.387,166.679,51.600,159.409
C05367=1020.507,8.651,397.373,166.682,51.594,159.408
C05368=1020.513,8.900,397.358,166.686,51.589,159.408
C05369=1020.518,9.150,397.344,166.687,51.584,159.407
C05370=1020.524,9.399,397.330,166.690,51.578,159.407
C05371=1020.531,9.649,397.316,166.694,51.573,159.406
C05372=1020.536,9.898,397.302,166.696,51.568,159.406
C05373=1020.542,10.148,397.288,166.698,51.562,159.405
C05374=1020.547,10.398,397.274,166.702,51.557,159.405
C05375=1020.554,10.680,397.258,166.704,51.551,159.404
C05376=1020.561,10.962,397.242,166.707,51.545,159.404
C05377=1020.568,11.245,397.226,166.711,51.539,159.403
C05378=1020.574,11.528,397.210,166.714,51.533,159.403
C05379=1020.580,11.777,397.196,166.717,51.528,159.402
C05380=1020.585,12.026,397.182,166.719,51.522,159.401
C05381=1020.591,12.276,397.168,166.722,51.517,159.401
C05382=1020.598,12.525,397.154,166.725,51.512,159.401
C05383=1020.603,12.775,397.140,166.727,51.506,159.400
C05384=1020.609,13.025,397.126,166.730,51.501,159.399
C05385=1020.615,13.274,397.111,166.733,51.496,159.399
C05386=1020.621,13.523,397.097,166.735,51.491,159.398
C05387=1020.627,13.773,397.082,166.738,51.485,159.398
C05388=1020.633,14.023,397.068,166.741,51.480,159.397
C05389=1020.638,14.272,397.054,166.743,51.475,159.397
C05390=1020.644,14.522,397.039,166.746,51.469,159.397
C05391=1020.649,14.771,397.024,166.748,51.465,159.396
C05392=1020.655,15.021,397.011,166.751,51.459,159.395
C05393=1020.661,15.270,396.996,166.754,51.453,159.395
C05394=1020.667,15.519,396.981,166.756,51.448,159.394
C05395=1020.673,15.769,396.967,166.760,51.443,159.394
C05396=1020.679,16.019,396.952,166.762,51.438,159.393
C05397=1020.684,16.269,396.938,166.764,51.432,159.393
C05398=1020.689,16.517,396.923,166.768,51.427,159.392
C05399=1020.696,16.768,396.909,166.770,51.422,159.392
C05400=1020.701,17.017,396.894,166.773,51.417,159.392
C05401=1020.708,17.266,396.879,166.776,51.411,159.391
C05402=1020.713,17.516,396.866,166.778,51.406,159.390
C05403=1020.719,17.765,396.851,166.781,51.401,159.390
C05404=1020.725,18.015,396.837,166.783,51.396,159.389
C05405=1020.730,18.264,396.822,166.786,51.390,159.389
C05406=1020.736,18.514,396.807,166.789,51.385,159.388
C05407=1020.742,18.764,396.793,166.791,51.380,159.388
C05408=1020.748,19.013,396.778,166.794,51.374,159.387
C05409=1020.754,19.262,396.763,166.797,51.369,159.387
C05410=1020.759,19.512,396.749,166.799,51.364,159.386
C05411=1020.765,19.762,396.734,166.802,51.359,159.386
C05412=1020.771,20.011,396.719,166.804,51.354,159.385
C05413=1020.776,20.260,396.705,166.807,51.348,159.385
C05414=1020.782,20.510,396.690,166.809,51.343,159.384
C05415=1020.788,20.759,396.675,166.813,51.338,159.384
C05416=1020.794,21.009,396.660,166.816,51.333,159.383
C05417=1020.799,21.259,396.646,166.817,51.327,159.383
C05418=1020.805,21.508,396.631,166.821,51.322,159.382
C05419=1020.811,21.757,396.616,166.823,51.317,159.382
C05420=1020.817,22.006,396.602,166.826,51.312,159.381
C05421=1020.823,22.256,396.586,166.829,51.306,159.381
C05422=1020.828,22.506,396.572,166.831,51.301,159.380
C05423=1020.834,22.756,396.557,166.834,51.296,159.380
C05424=1020.840,23.005,396.542,166.836,51.291,159.379
C05425=1020.846,23.255,396.527,166.839,51.285,159.379
C05426=1020.852,23.503,396.513,166.842,51.280,159.378
C05427=1020.857,23.754,396.498,166.844,51.275,159.378
C05428=1020.863,24.003,396.483,166.847,51.269,159.377
C05429=1020.869,24.253,396.468,166.849,51.265,159.376
C05430=1020.875,24.502,396.454,166.852,51.259,159.376
C05431=1020.881,24.752,396.438,166.855,51.253,159.375
C05432=1020.886,25.001,396.424,166.857,51.249,159.375
C05433=1020.893,25.250,396.409,166.861,51.243,159.375
C05434=1020.898,25.500,396.394,166.863,51.237,159.374
C05435=1020.904,25.750,396.379,166.865,51.233,159.373
C05436=1020.910,25.999,396.365,166.869,51.227,159.373
C05437=1020.915,26.249,396.349,166.870,51.222,159.372
C05438=1020.921,26.498,396.335,166.874,51.217,159.372
C05439=1020.928,26.782,396.317,166.876,51.211,159.371
C05440=1020.934,27.066,396.300,166.879,51.205,159.371
C05441=1020.941,27.350,396.283,166.883,51.199,159.370
C05442=1020.948,27.634,396.266,166.886,51.193,159.369
C05443=1020.953,27.883,396.252,166.889,51.187,159.369
C05444=1020.959,28.133,396.236,166.891,51.182,159.368
C05445=1020.965,28.382,396.221,166.894,51.177,159.368
C05446=1020.971,28.632,396.206,166.896,51.172,159.367
C05447=1020.976,28.881,396.191,166.899,51.166,159.367
C05448=1020.982,29.131,396.176,166.901,51.161,159.366
C05449=1020.988,29.380,396.161,166.904,51.156,159.366
C05450=1020.994,29.629,396.145,166.906,51.151,159.365
C05451=1020.999,29.879,396.129,166.909,51.145,159.365
C05452=1021.005,30.128,396.115,166.912,51.140,159.364
